// TIA Portal V20 export
// export: Created 2025-12-01T14:57:42.0271805Z, ExportSetting None, DisplayName Totally Integrated Automation Portal, DisplayVersion V20 Update 3, DisplayName TIA Portal Openness, DisplayVersion V20 Update 3, DisplayName TIA Portal Version Control Interface, DisplayVersion V20 Update 3, DisplayName STEP 7 Professional, DisplayVersion V20 Update 3, DisplayName STEP 7 Safety, DisplayVersion V20 Update 2, DisplayName WinCC Basic/Comfort/Advanced, DisplayVersion V20 Update 3, DisplayName WinCC Professional, DisplayVersion V20 Update 3, DisplayName WinCC Unified, DisplayVersion V20 Update 3
FUNCTION_BLOCK "FB382_HorquillaLenze_Paletizador_NDD_E3S3"   // FB382, LAD
{ S7_Optimized_Access := 'FALSE' }
// stored: AutoNumber false, SetENOAutomatically false
   VAR_INPUT
      Mesa : UInt;   // Mesa de la FB
      NDB_ConfigNDD : UInt;   // DB de Configuracion General del NDD
      NDB_DatosNDD : UInt;   // DB de Configuracion Particular del NDD
      OffsetDatosHorquilla : UInt;   // Offset de los datos particulares de la Horquilla
      DesHabilitar_Horq : Bool;   // DesHabilitar la Horquilla
      Mantenimiento : Bool;   // En Mantenimiento la Horquilla
      Error_Tx : Bool;   // Error de la Zona
      EnTension : Bool;   // Existe Tension en la Mesa
      TermicoFreno_Horq : Bool;   // Termico del Freno de la Horquilla
      Horq_PresCarga : Bool;   // Presencia de Carga en la Horquilla
      Horq_Protusion : Bool;
      Horq_SeguridadUp_Libre : Bool;
      Horq_SeguridadUp_Ocupada : Bool;
      Horq_SeguridadDown : Bool;
      BarreraNivelDown : Bool;
      EM_Horq_Out : Bool;   // Emergencia al Recoger la Horquilla
      Horq_Out : Bool;   // Horquilla Recogida
      Horq_In : Bool;   // Horquilla Fuera (En el Elevador)
      EM_Horq_In : Bool;   // Emergencia al Extender la Horquilla
      Manual_HorqIn : Bool;   // Extender la Horquilla en Manual
      Manual_HorqOut : Bool;   // Recoger la Horquilla en Manual
      Homming_Horq : Bool;   // Realizar el Homing del Variador de la Horquilla (RefCero >> Out)
      pHsRef_Horq : Bool;
      F_EnvMens_PMx : Bool;
      V_TOut_Horquilla : Time := T#5s;   // Valor de Time Out del Movimiento de la Horquilla
      V_TOut_Protusion : Time := T#500ms;
   END_VAR
   VAR_OUTPUT
      P_EnvMens_PMx : Bool;
   END_VAR
   VAR_IN_OUT
      Interlock_Horquilla : "NDD_Interlock_Horquilla";
   END_VAR
   VAR
      TOut_Horquilla { S7_SetPoint := 'True'} : TON_TIME;   // Time Out del Moviento de la Hoquilla
      TOut_Protusion { S7_SetPoint := 'True'} : TON_TIME;
      TEstableMovHorq { S7_SetPoint := 'True'} : TON_TIME;
      TEsperaMoverHorq { S7_SetPoint := 'True'} : TON_TIME;
      MemoPosicionActual_Horq : Int;
      PosicionActual_Horq : Int;   // Posicion Actual de la Horquilla (Variador)
      PosicionOut_Horq : Int;   // Posicion Out de la Horquilla (DB del NDD)
      PosicionIn_Horq { ExternalVisible := 'False'} : Int;   // Posicion In de la Horquilla (DB del NDD)
      PosicionMover_Horq : Int;
      ConsignaFR_Horq : Int;
      SubjectArea_Horq : Word;
      IDArea_Horq : Word;
      NodoNoPres_VarHorq : Bool;   // Nodo del Variador de la Horquilla - No presente
      MoverHorq : Bool;
      FinMoverHorq : Bool;
      MemoFinMorverHorq : Bool;
      PosHorqOut_OK : Bool;   // La Hoquilla esta en Reposo, esta en OUT
      PosHorqIn_OK : Bool;
      MA_Horquilla_IN : Bool;
      MA_Horquilla_OUT : Bool;
      HORQ_ET00 : Bool;   // Etapas de la Horquilla
      HORQ_ET01 : Bool;   // Etapas de la Horquilla
      HORQ_RST01 : Bool;   // Etapas de la Horquilla
      HORQ_RST02 : Bool;   // Etapas de la Horquilla
      HORQ_CAR01 : Bool;   // Etapas de la Horquilla
      HORQ_CAR02 : Bool;   // Etapas de la Horquilla
      HORQ_CAR03 : Bool;   // Etapas de la Horquilla
      HORQ_CAR04 : Bool;
      HORQ_ET02 : Bool;   // Etapas de la Horquilla
      HORQ_DCAR01 : Bool;   // Etapas de la Horquilla
      HORQ_DCAR02 : Bool;   // Etapas de la Horquilla
      HORQ_DCAR03 : Bool;   // Etapas de la Horquilla
      HORQ_DCAR04 : Bool;
      STAT_P_EnvMens_PMx : Bool;
      ErrorVar_Horquilla : Bool;
      ReferenciaOK_Horq : Bool;
      MemoReferenciaOK_Horq : Bool;
      MemoHoming_Horq : Bool;
   END_VAR
   VAR_TEMP
      EstadoZona : "EstadoZona";
      EstadoVI : "EstadosMesa_HorquillaLenze_Paletizador_NDD";
      NodoVar_Horq : "Status_NodosProfinet";
      Guardar_AR1 : DWord;
      Guardar_AR2 : DWord;
      P_DatosHorquilla : DWord;   // Puntero a los datos de la Horquilla (Configuracionn del Paletizador)
      P_NodoVar_Horq : DWord;
      DB_ConfigNDD : Word;   // DB de Configuracion General de los NDD
      DB_DatosNDD : Word;   // DB del NDD (Configuracion del Paletizador)
      NumDB_DiagProfinet : Word;
      NumNodo_VarHorq : Int;
      ByteInicial_VarHorq : Int;
      VeloManual_Horq : Int;   // Velocidad Manual
      VeloRapidaOut_Horq : Int;   // Velocidad Rapida para ir a Posicion Out
      VeloLentaOut_Horq : Int;   // Velocidad Lenta para ir a Posicion Out
      PosLentaOut_Horq : Int;   // Diferencia para pasar Lenta para ir a Posicion Out
      VeloRapidaIn_Horq : Int;   // Velocidad Rapida para ir a Posicion In
      VeloLentaIn_Horq : Int;   // Velocidad Lenta para ir a Posicion In
      PosLentaIn_Horq : Int;   // Diferencia para pasar Lenta para ir a Posicion In
      AuxMargen : Int;
      AuxPosMax : Int;
      AuxPosMin : Int;
      TempInt : Int;
      AuxEstados : Bool;
      DestinoHorq_OUT : Bool;
      DestinoHorq_IN : Bool;
      MoverHorq_LentaOUT : Bool;
      MoverHorq_LentaIN : Bool;
   END_VAR
   VAR_TEMP   // added for the SCL form of the ladder/FBD networks
      _w1 : Bool;
      _w2 : Bool;
      _w3 : Bool;
   END_VAR
BEGIN

REGION Network 1: INICIALIZACIONES
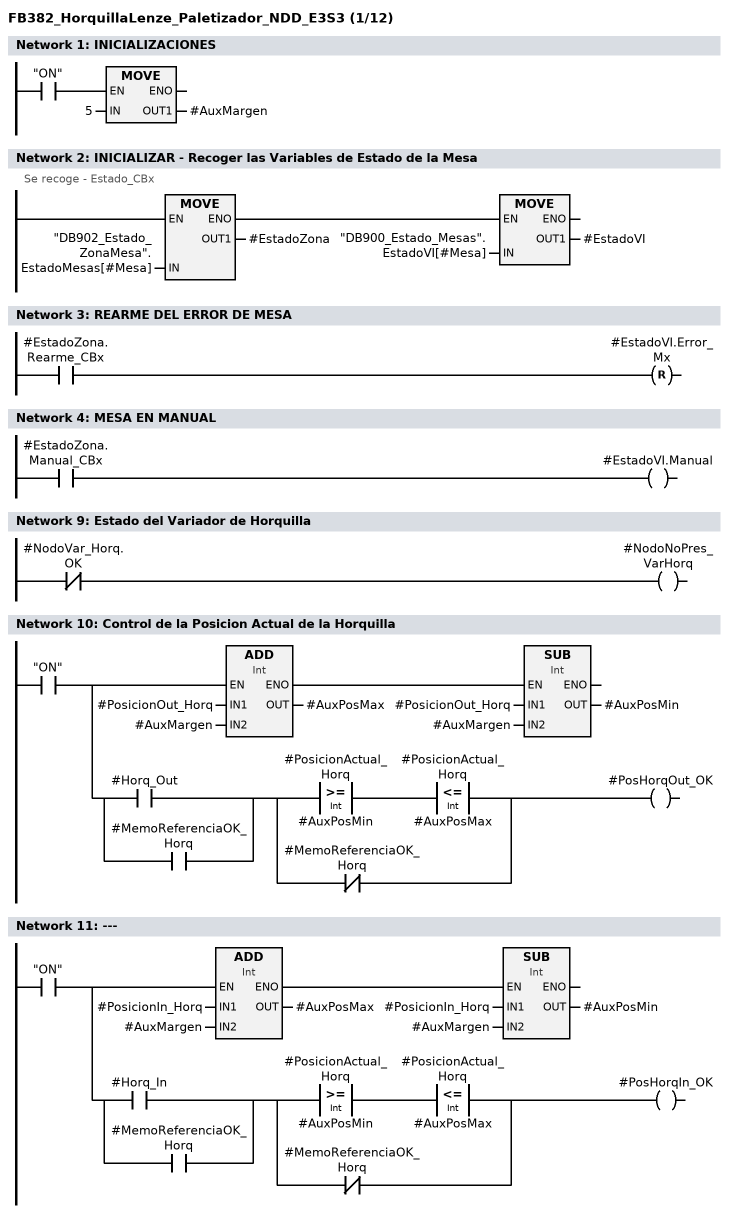
   RUNG wire#powerrail
      Contact( "ON" )
      { S7_GenerateENO := "TRUE" } Move(in := 5, out1 => #AuxMargen)
   END_RUNG
   // the same network as SCL:
   IF "ON" THEN #AuxMargen := 5; END_IF;
END_REGION

REGION Network 2: INICIALIZAR - Recoger las Variables de Estado de la Mesa
   // Se recoge - Estado_CBx
   RUNG wire#powerrail
      Move(in := "DB902_Estado_ZonaMesa".EstadoMesas[#Mesa], out1 => #EstadoZona)
      Move(in := "DB900_Estado_Mesas".EstadoVI[#Mesa], out1 => #EstadoVI)
   END_RUNG
   // the same network as SCL:
   #EstadoZona := "DB902_Estado_ZonaMesa".EstadoMesas[#Mesa];
   #EstadoVI := "DB900_Estado_Mesas".EstadoVI[#Mesa];
END_REGION

REGION Network 3: REARME DEL ERROR DE MESA
   RUNG wire#powerrail
      Contact( #EstadoZona.Rearme_CBx )
      R_Coil( #EstadoVI.Error_Mx )
   END_RUNG
   // the same network as SCL:
   IF #EstadoZona.Rearme_CBx THEN #EstadoVI.Error_Mx := FALSE; END_IF;
END_REGION

REGION Network 4: MESA EN MANUAL
   RUNG wire#powerrail
      Contact( #EstadoZona.Manual_CBx )
      Coil( #EstadoVI.Manual )
   END_RUNG
   // the same network as SCL:
   #EstadoVI.Manual := #EstadoZona.Manual_CBx;
END_REGION

NETWORK
TITLE = Datos Internos de la Horquilla
// ------------------------------------------------------------------------------------
// ------------------------------------------------------------------------------------
// --- Previas

      TAR1  #Guardar_AR1;  // Guardar AR1 y AR2


// ------------------------------------------------------------------------------------
// ------------------------------------------------------------------------------------
// --- Datos iniciales

      L     #NDB_DatosNDD;  // - DB del Paletizador NDD
      T     #DB_DatosNDD;

      L     #NDB_ConfigNDD;  // - DB del Config de los Paletizadores MDD
      T     #DB_ConfigNDD;  //

      L     #OffsetDatosHorquilla;  // Puntero a los Datos de Horquilla
      SLD   3;
      T     #P_DatosHorquilla;


/////////////////////////////////////////////////////////////////////////////
/////////////////////////////////////////////////////////////////////////////
// --- Sistema de Profinet

      LAR1  P#0.0;  // - Leer Datos de los Variadores
      OPN   DB [#DB_DatosNDD];  //   del NDD

      L     DBW [AR1, P#0.0];  // - Num DB de Profinet
      T     #NumDB_DiagProfinet;
      L     DBW [AR1, P#6.0];  // - Nodos de los Variadores
      T     #NumNodo_VarHorq;
      L     DBW [AR1, P#12.0];  // - Direcciones de los Variadores
      T     #ByteInicial_VarHorq;

      L     P##NodoVar_Horq;  // Puntero del Estado del Nodo del Variador de Horquilla (TEMPORAL)
      T     #P_NodoVar_Horq;



NETWORK
TITLE = ---
// ------------------------------------------------------------------------------------
// ------------------------------------------------------------------------------------
// --- Datos Generales de Configuracion de los NDD

      LAR1  P#0.0;  // - Leer Datos de Velocidad de la Horquilla
      OPN   DB [#DB_ConfigNDD];

      L     DBW [AR1, P#16.0];  // - Velocidad en Manual
      T     #VeloManual_Horq;

      L     DBW [AR1, P#18.0];  // - Velocidad del Mov. hacia In
      T     #VeloRapidaIn_Horq;
      L     DBW [AR1, P#20.0];
      T     #VeloLentaIn_Horq;

      L     DBW [AR1, P#22.0];  // - Velocidad del Mov. hacia Out
      T     #VeloRapidaOut_Horq;
      L     DBW [AR1, P#24.0];
      T     #VeloLentaOut_Horq;

      L     DBW [AR1, P#26.0];  // - Posiciones de Cambio de Velocidad
      T     #PosLentaIn_Horq;
      L     DBW [AR1, P#28.0];
      T     #PosLentaOut_Horq;



NETWORK
TITLE = ----
// ------------------------------------------------------------------------------------
// ------------------------------------------------------------------------------------
// --- Datos Particulares de la Horquilla del NDD

      LAR1  #P_DatosHorquilla;  // - Leer Datos de la Horquilla
      OPN   DB [#DB_DatosNDD];
      L     DBW [AR1, P#0.0];
      T     #PosicionIn_Horq;
      L     DBW [AR1, P#2.0];
      T     #PosicionOut_Horq;


// ------------------------------------------------------------------------------------
// ------------------------------------------------------------------------------------
// --- Estado del Nodo de PROFINET del Variador de la Horquilla (LENZE)

      L     #NumNodo_VarHorq;  // Nodo de Profinet
      L     1;
      -I;
      L     2;  // Longitud registro datos
      *I;
      SLD   3;
      LAR1;

      OPN   DB [#NumDB_DiagProfinet];  // Leer estado del Nodo de PROFINET
      L     DBW [AR1, P#0.0];
      T     LW [#P_NodoVar_Horq];




NETWORK
TITLE = ---
// ------------------------------------------------------------------------------------
// ------------------------------------------------------------------------------------
// --- Final de Datos Inicialies

      LAR1  #Guardar_AR1;  // Recuperar AR1 y AR2



REGION Network 9: Estado del Variador de Horquilla
   RUNG wire#powerrail
      I_Contact( #NodoVar_Horq.OK )
      Coil( #NodoNoPres_VarHorq )
   END_RUNG
   // the same network as SCL:
   #NodoNoPres_VarHorq := NOT #NodoVar_Horq.OK;
END_REGION

REGION Network 10: Control de la Posicion Actual de la Horquilla
   RUNG wire#powerrail
      Contact( "ON" )
      wire#w1
      { S7_Templates := "SrcType := Int"; S7_GenerateENO := "TRUE" } Add(in1 := #PosicionOut_Horq, in2 := #AuxMargen, out => #AuxPosMax)
      { S7_Templates := "SrcType := Int"; S7_GenerateENO := "TRUE" } Sub(in1 := #PosicionOut_Horq, in2 := #AuxMargen, out => #AuxPosMin)
   END_RUNG
   RUNG wire#w1
      Contact( #Horq_Out )
      wire#w2
      { S7_Templates := "SrcType := Int" } GE_Contact(in1 := #PosicionActual_Horq, in2 := #AuxPosMin)
      { S7_Templates := "SrcType := Int" } LE_Contact(in1 := #PosicionActual_Horq, in2 := #AuxPosMax)
      wire#w3
      Coil( #PosHorqOut_OK )
   END_RUNG
   RUNG wire#w1
      Contact( #MemoReferenciaOK_Horq )
   END_RUNG wire#w2
   RUNG wire#w2
      I_Contact( #MemoReferenciaOK_Horq )
   END_RUNG wire#w3
   // the same network as SCL:
   // ENO of a box is taken as its EN; it also drops when the box reports an error
   IF "ON" THEN
       #AuxPosMax := #PosicionOut_Horq + #AuxMargen;
       #AuxPosMin := #PosicionOut_Horq - #AuxMargen;
   END_IF;
   #PosHorqOut_OK := "ON" AND (#Horq_Out OR #MemoReferenciaOK_Horq) AND (((#PosicionActual_Horq >= #AuxPosMin) AND (#PosicionActual_Horq <= #AuxPosMax)) OR NOT #MemoReferenciaOK_Horq);
END_REGION

REGION Network 11: ---
   RUNG wire#powerrail
      Contact( "ON" )
      wire#w1
      { S7_Templates := "SrcType := Int"; S7_GenerateENO := "TRUE" } Add(in1 := #PosicionIn_Horq, in2 := #AuxMargen, out => #AuxPosMax)
      { S7_Templates := "SrcType := Int"; S7_GenerateENO := "TRUE" } Sub(in1 := #PosicionIn_Horq, in2 := #AuxMargen, out => #AuxPosMin)
   END_RUNG
   RUNG wire#w1
      Contact( #Horq_In )
      wire#w2
      { S7_Templates := "SrcType := Int" } GE_Contact(in1 := #PosicionActual_Horq, in2 := #AuxPosMin)
      { S7_Templates := "SrcType := Int" } LE_Contact(in1 := #PosicionActual_Horq, in2 := #AuxPosMax)
      wire#w3
      Coil( #PosHorqIn_OK )
   END_RUNG
   RUNG wire#w1
      Contact( #MemoReferenciaOK_Horq )
   END_RUNG wire#w2
   RUNG wire#w2
      I_Contact( #MemoReferenciaOK_Horq )
   END_RUNG wire#w3
   // the same network as SCL:
   // ENO of a box is taken as its EN; it also drops when the box reports an error
   IF "ON" THEN
       #AuxPosMax := #PosicionIn_Horq + #AuxMargen;
       #AuxPosMin := #PosicionIn_Horq - #AuxMargen;
   END_IF;
   #PosHorqIn_OK := "ON" AND (#Horq_In OR #MemoReferenciaOK_Horq) AND (((#PosicionActual_Horq >= #AuxPosMin) AND (#PosicionActual_Horq <= #AuxPosMax)) OR NOT #MemoReferenciaOK_Horq);
END_REGION

REGION Network 12: ---
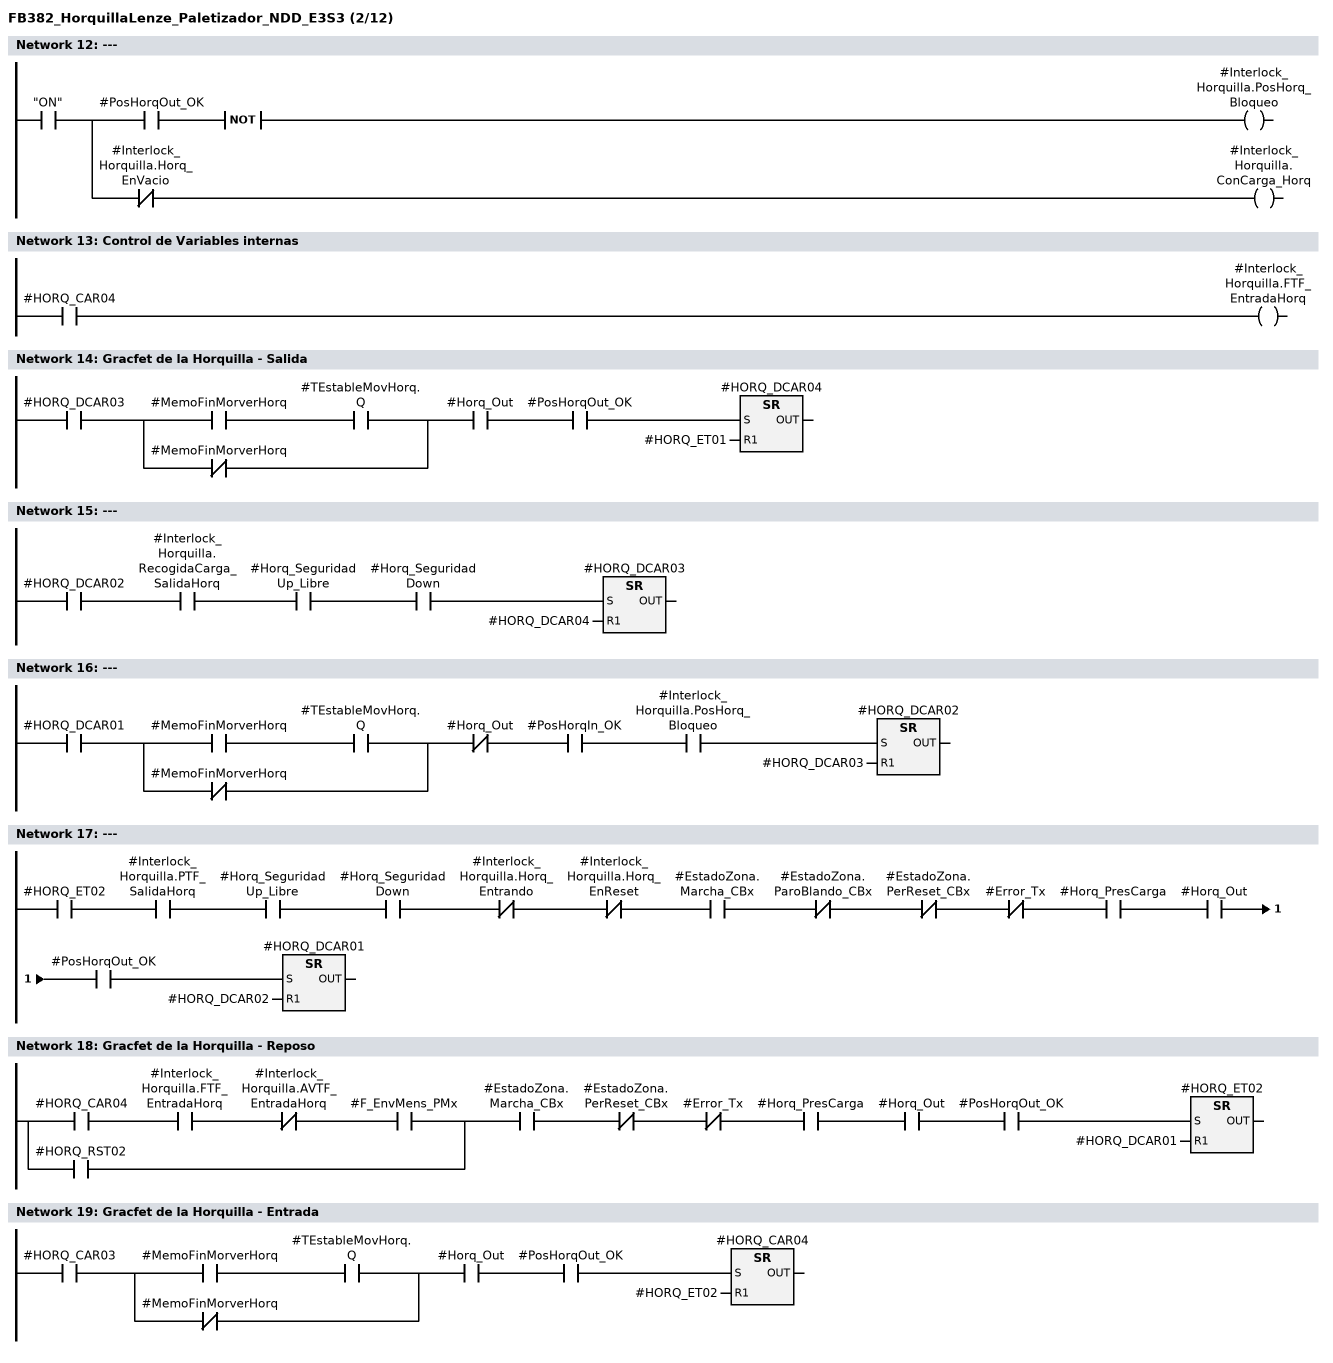
   RUNG wire#powerrail
      Contact( "ON" )
      wire#w1
      Contact( #PosHorqOut_OK )
      Not()
      Coil( #Interlock_Horquilla.PosHorq_Bloqueo )
   END_RUNG
   RUNG wire#w1
      I_Contact( #Interlock_Horquilla.Horq_EnVacio )
      Coil( #Interlock_Horquilla.ConCarga_Horq )
   END_RUNG
   // the same network as SCL:
   #Interlock_Horquilla.PosHorq_Bloqueo := NOT ("ON" AND #PosHorqOut_OK);
   #Interlock_Horquilla.ConCarga_Horq := "ON" AND NOT #Interlock_Horquilla.Horq_EnVacio;
END_REGION

REGION Network 13: Control de Variables internas
   RUNG wire#powerrail
      Contact( #HORQ_CAR04 )
      Coil( #Interlock_Horquilla.FTF_EntradaHorq )
   END_RUNG
   // the same network as SCL:
   #Interlock_Horquilla.FTF_EntradaHorq := #HORQ_CAR04;
END_REGION

REGION Network 14: Gracfet de la Horquilla - Salida
   RUNG wire#powerrail
      Contact( #HORQ_DCAR03 )
      wire#w1
      Contact( #MemoFinMorverHorq )
      Contact( #TEstableMovHorq.Q )
      wire#w2
      Contact( #Horq_Out )
      Contact( #PosHorqOut_OK )
      S_SR(operand := #HORQ_DCAR04, r1 := #HORQ_ET01)
   END_RUNG
   RUNG wire#w1
      I_Contact( #MemoFinMorverHorq )
   END_RUNG wire#w2
   // the same network as SCL:
   IF #HORQ_DCAR03 AND ((#MemoFinMorverHorq AND #TEstableMovHorq.Q) OR NOT #MemoFinMorverHorq) AND #Horq_Out AND #PosHorqOut_OK THEN
       #HORQ_DCAR04 := TRUE;   // SR flip-flop
   END_IF;
   IF #HORQ_ET01 THEN #HORQ_DCAR04 := FALSE; END_IF;
END_REGION

REGION Network 15: ---
   RUNG wire#powerrail
      Contact( #HORQ_DCAR02 )
      Contact( #Interlock_Horquilla.RecogidaCarga_SalidaHorq )
      Contact( #Horq_SeguridadUp_Libre )
      Contact( #Horq_SeguridadDown )
      S_SR(operand := #HORQ_DCAR03, r1 := #HORQ_DCAR04)
   END_RUNG
   // the same network as SCL:
   IF #HORQ_DCAR02 AND #Interlock_Horquilla.RecogidaCarga_SalidaHorq AND #Horq_SeguridadUp_Libre AND #Horq_SeguridadDown THEN
       #HORQ_DCAR03 := TRUE;   // SR flip-flop
   END_IF;
   IF #HORQ_DCAR04 THEN #HORQ_DCAR03 := FALSE; END_IF;
END_REGION

REGION Network 16: ---
   RUNG wire#powerrail
      Contact( #HORQ_DCAR01 )
      wire#w1
      Contact( #MemoFinMorverHorq )
      Contact( #TEstableMovHorq.Q )
      wire#w2
      I_Contact( #Horq_Out )
      Contact( #PosHorqIn_OK )
      Contact( #Interlock_Horquilla.PosHorq_Bloqueo )
      S_SR(operand := #HORQ_DCAR02, r1 := #HORQ_DCAR03)
   END_RUNG
   RUNG wire#w1
      I_Contact( #MemoFinMorverHorq )
   END_RUNG wire#w2
   // the same network as SCL:
   IF #HORQ_DCAR01 AND ((#MemoFinMorverHorq AND #TEstableMovHorq.Q) OR NOT #MemoFinMorverHorq) AND NOT #Horq_Out AND #PosHorqIn_OK AND #Interlock_Horquilla.PosHorq_Bloqueo THEN
       #HORQ_DCAR02 := TRUE;   // SR flip-flop
   END_IF;
   IF #HORQ_DCAR03 THEN #HORQ_DCAR02 := FALSE; END_IF;
END_REGION

REGION Network 17: ---
   RUNG wire#powerrail
      Contact( #HORQ_ET02 )
      Contact( #Interlock_Horquilla.PTF_SalidaHorq )
      Contact( #Horq_SeguridadUp_Libre )
      Contact( #Horq_SeguridadDown )
      I_Contact( #Interlock_Horquilla.Horq_Entrando )
      I_Contact( #Interlock_Horquilla.Horq_EnReset )
      Contact( #EstadoZona.Marcha_CBx )
      I_Contact( #EstadoZona.ParoBlando_CBx )
      I_Contact( #EstadoZona.PerReset_CBx )
      I_Contact( #Error_Tx )
      Contact( #Horq_PresCarga )
      Contact( #Horq_Out )
      Contact( #PosHorqOut_OK )
      S_SR(operand := #HORQ_DCAR01, r1 := #HORQ_DCAR02)
   END_RUNG
   // the same network as SCL:
   IF #HORQ_ET02 AND #Interlock_Horquilla.PTF_SalidaHorq AND #Horq_SeguridadUp_Libre AND #Horq_SeguridadDown AND NOT #Interlock_Horquilla.Horq_Entrando AND NOT #Interlock_Horquilla.Horq_EnReset AND #EstadoZona.Marcha_CBx AND NOT #EstadoZona.ParoBlando_CBx AND NOT #EstadoZona.PerReset_CBx AND NOT #Error_Tx AND #Horq_PresCarga AND #Horq_Out AND #PosHorqOut_OK THEN
       #HORQ_DCAR01 := TRUE;   // SR flip-flop
   END_IF;
   IF #HORQ_DCAR02 THEN #HORQ_DCAR01 := FALSE; END_IF;
END_REGION

REGION Network 18: Gracfet de la Horquilla - Reposo
   RUNG wire#powerrail
      Contact( #HORQ_CAR04 )
      Contact( #Interlock_Horquilla.FTF_EntradaHorq )
      I_Contact( #Interlock_Horquilla.AVTF_EntradaHorq )
      Contact( #F_EnvMens_PMx )
      wire#w1
      Contact( #EstadoZona.Marcha_CBx )
      I_Contact( #EstadoZona.PerReset_CBx )
      I_Contact( #Error_Tx )
      Contact( #Horq_PresCarga )
      Contact( #Horq_Out )
      Contact( #PosHorqOut_OK )
      S_SR(operand := #HORQ_ET02, r1 := #HORQ_DCAR01)
   END_RUNG
   RUNG wire#powerrail
      Contact( #HORQ_RST02 )
   END_RUNG wire#w1
   // the same network as SCL:
   IF ((#HORQ_CAR04 AND #Interlock_Horquilla.FTF_EntradaHorq AND NOT #Interlock_Horquilla.AVTF_EntradaHorq AND #F_EnvMens_PMx) OR #HORQ_RST02) AND #EstadoZona.Marcha_CBx AND NOT #EstadoZona.PerReset_CBx AND NOT #Error_Tx AND #Horq_PresCarga AND #Horq_Out AND #PosHorqOut_OK THEN
       #HORQ_ET02 := TRUE;   // SR flip-flop
   END_IF;
   IF #HORQ_DCAR01 THEN #HORQ_ET02 := FALSE; END_IF;
END_REGION

REGION Network 19: Gracfet de la Horquilla - Entrada
   RUNG wire#powerrail
      Contact( #HORQ_CAR03 )
      wire#w1
      Contact( #MemoFinMorverHorq )
      Contact( #TEstableMovHorq.Q )
      wire#w2
      Contact( #Horq_Out )
      Contact( #PosHorqOut_OK )
      S_SR(operand := #HORQ_CAR04, r1 := #HORQ_ET02)
   END_RUNG
   RUNG wire#w1
      I_Contact( #MemoFinMorverHorq )
   END_RUNG wire#w2
   // the same network as SCL:
   IF #HORQ_CAR03 AND ((#MemoFinMorverHorq AND #TEstableMovHorq.Q) OR NOT #MemoFinMorverHorq) AND #Horq_Out AND #PosHorqOut_OK THEN
       #HORQ_CAR04 := TRUE;   // SR flip-flop
   END_IF;
   IF #HORQ_ET02 THEN #HORQ_CAR04 := FALSE; END_IF;
END_REGION

REGION Network 20: ---
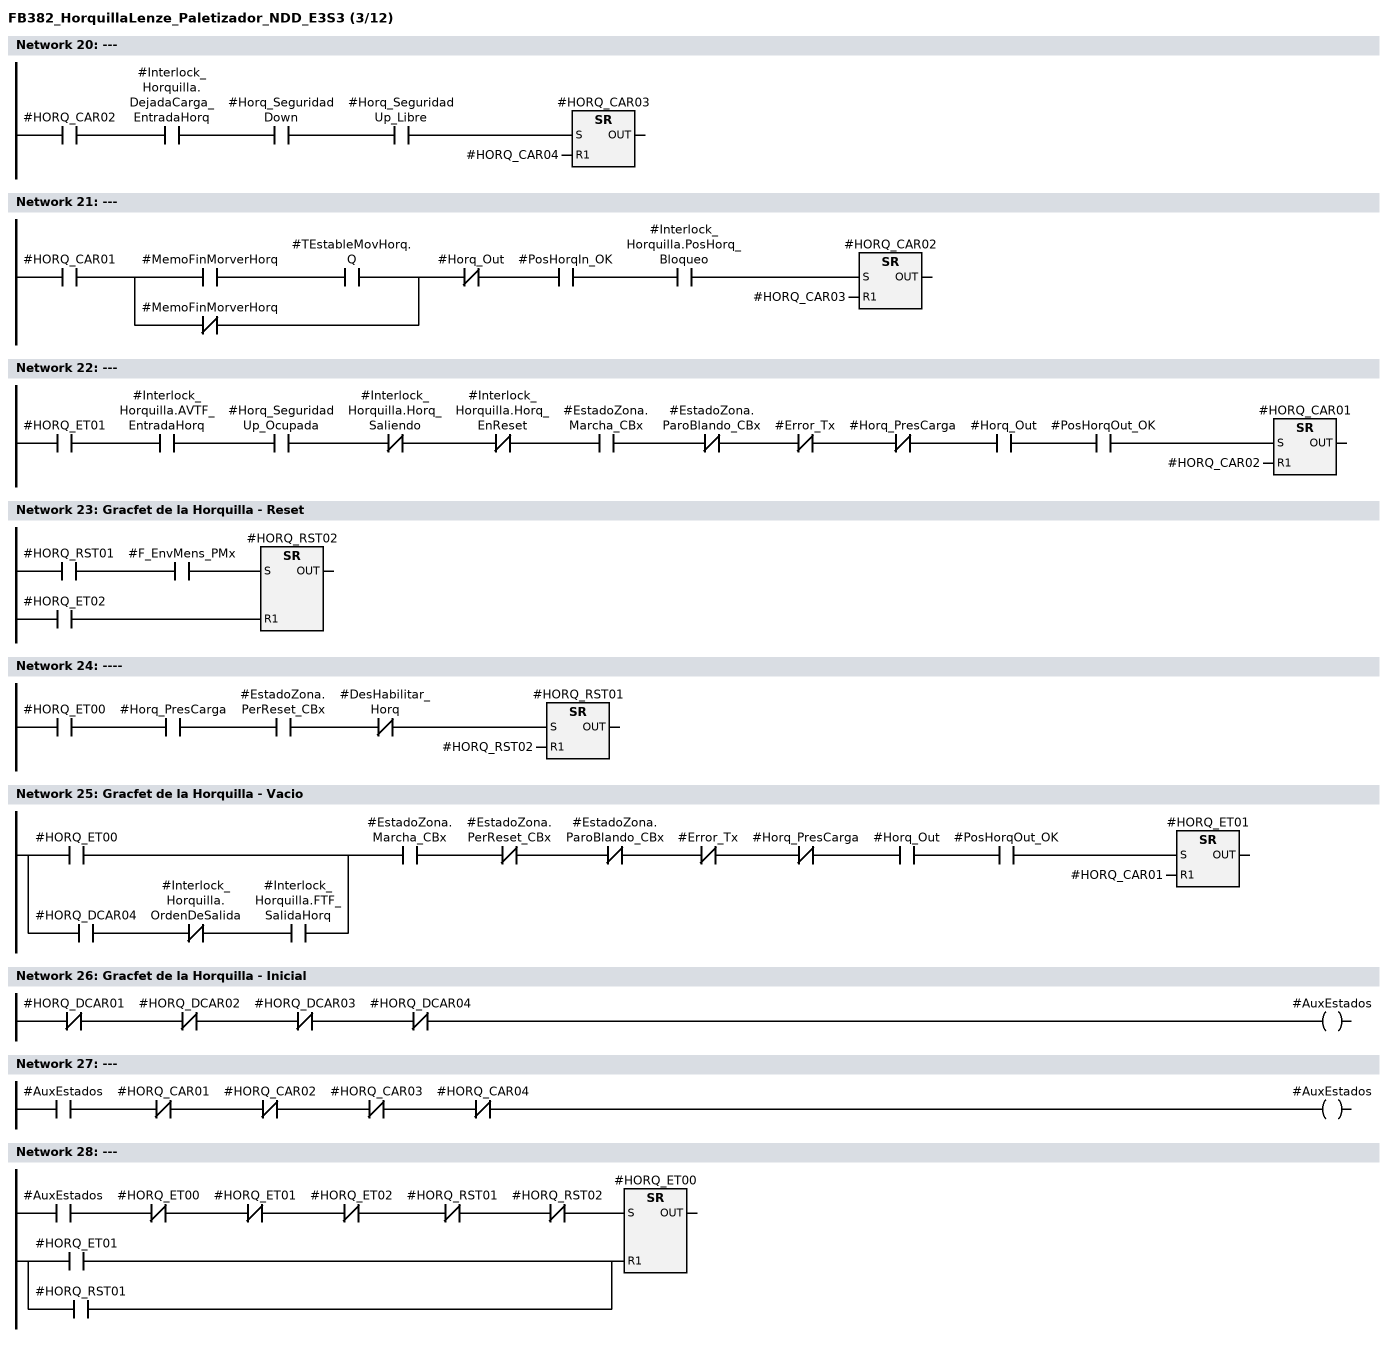
   RUNG wire#powerrail
      Contact( #HORQ_CAR02 )
      Contact( #Interlock_Horquilla.DejadaCarga_EntradaHorq )
      Contact( #Horq_SeguridadDown )
      Contact( #Horq_SeguridadUp_Libre )
      S_SR(operand := #HORQ_CAR03, r1 := #HORQ_CAR04)
   END_RUNG
   // the same network as SCL:
   IF #HORQ_CAR02 AND #Interlock_Horquilla.DejadaCarga_EntradaHorq AND #Horq_SeguridadDown AND #Horq_SeguridadUp_Libre THEN
       #HORQ_CAR03 := TRUE;   // SR flip-flop
   END_IF;
   IF #HORQ_CAR04 THEN #HORQ_CAR03 := FALSE; END_IF;
END_REGION

REGION Network 21: ---
   RUNG wire#powerrail
      Contact( #HORQ_CAR01 )
      wire#w1
      Contact( #MemoFinMorverHorq )
      Contact( #TEstableMovHorq.Q )
      wire#w2
      I_Contact( #Horq_Out )
      Contact( #PosHorqIn_OK )
      Contact( #Interlock_Horquilla.PosHorq_Bloqueo )
      S_SR(operand := #HORQ_CAR02, r1 := #HORQ_CAR03)
   END_RUNG
   RUNG wire#w1
      I_Contact( #MemoFinMorverHorq )
   END_RUNG wire#w2
   // the same network as SCL:
   IF #HORQ_CAR01 AND ((#MemoFinMorverHorq AND #TEstableMovHorq.Q) OR NOT #MemoFinMorverHorq) AND NOT #Horq_Out AND #PosHorqIn_OK AND #Interlock_Horquilla.PosHorq_Bloqueo THEN
       #HORQ_CAR02 := TRUE;   // SR flip-flop
   END_IF;
   IF #HORQ_CAR03 THEN #HORQ_CAR02 := FALSE; END_IF;
END_REGION

REGION Network 22: ---
   RUNG wire#powerrail
      Contact( #HORQ_ET01 )
      Contact( #Interlock_Horquilla.AVTF_EntradaHorq )
      Contact( #Horq_SeguridadUp_Ocupada )
      I_Contact( #Interlock_Horquilla.Horq_Saliendo )
      I_Contact( #Interlock_Horquilla.Horq_EnReset )
      Contact( #EstadoZona.Marcha_CBx )
      I_Contact( #EstadoZona.ParoBlando_CBx )
      I_Contact( #Error_Tx )
      I_Contact( #Horq_PresCarga )
      Contact( #Horq_Out )
      Contact( #PosHorqOut_OK )
      S_SR(operand := #HORQ_CAR01, r1 := #HORQ_CAR02)
   END_RUNG
   // the same network as SCL:
   IF #HORQ_ET01 AND #Interlock_Horquilla.AVTF_EntradaHorq AND #Horq_SeguridadUp_Ocupada AND NOT #Interlock_Horquilla.Horq_Saliendo AND NOT #Interlock_Horquilla.Horq_EnReset AND #EstadoZona.Marcha_CBx AND NOT #EstadoZona.ParoBlando_CBx AND NOT #Error_Tx AND NOT #Horq_PresCarga AND #Horq_Out AND #PosHorqOut_OK THEN
       #HORQ_CAR01 := TRUE;   // SR flip-flop
   END_IF;
   IF #HORQ_CAR02 THEN #HORQ_CAR01 := FALSE; END_IF;
END_REGION

REGION Network 23: Gracfet de la Horquilla - Reset
   RUNG wire#powerrail
      Contact( #HORQ_RST01 )
      Contact( #F_EnvMens_PMx )
      S_SR(operand := #HORQ_RST02, r1 := wire#w1)
   END_RUNG
   RUNG wire#powerrail
      Contact( #HORQ_ET02 )
   END_RUNG wire#w1
   // the same network as SCL:
   IF #HORQ_RST01 AND #F_EnvMens_PMx THEN
       #HORQ_RST02 := TRUE;   // SR flip-flop
   END_IF;
   IF #HORQ_ET02 THEN #HORQ_RST02 := FALSE; END_IF;
END_REGION

REGION Network 24: ----
   RUNG wire#powerrail
      Contact( #HORQ_ET00 )
      Contact( #Horq_PresCarga )
      Contact( #EstadoZona.PerReset_CBx )
      I_Contact( #DesHabilitar_Horq )
      S_SR(operand := #HORQ_RST01, r1 := #HORQ_RST02)
   END_RUNG
   // the same network as SCL:
   IF #HORQ_ET00 AND #Horq_PresCarga AND #EstadoZona.PerReset_CBx AND NOT #DesHabilitar_Horq THEN
       #HORQ_RST01 := TRUE;   // SR flip-flop
   END_IF;
   IF #HORQ_RST02 THEN #HORQ_RST01 := FALSE; END_IF;
END_REGION

REGION Network 25: Gracfet de la Horquilla - Vacio
   RUNG wire#powerrail
      Contact( #HORQ_ET00 )
      wire#w1
      Contact( #EstadoZona.Marcha_CBx )
      I_Contact( #EstadoZona.PerReset_CBx )
      I_Contact( #EstadoZona.ParoBlando_CBx )
      I_Contact( #Error_Tx )
      I_Contact( #Horq_PresCarga )
      Contact( #Horq_Out )
      Contact( #PosHorqOut_OK )
      S_SR(operand := #HORQ_ET01, r1 := #HORQ_CAR01)
   END_RUNG
   RUNG wire#powerrail
      Contact( #HORQ_DCAR04 )
      I_Contact( #Interlock_Horquilla.OrdenDeSalida )
      Contact( #Interlock_Horquilla.FTF_SalidaHorq )
   END_RUNG wire#w1
   // the same network as SCL:
   IF (#HORQ_ET00 OR (#HORQ_DCAR04 AND NOT #Interlock_Horquilla.OrdenDeSalida AND #Interlock_Horquilla.FTF_SalidaHorq)) AND #EstadoZona.Marcha_CBx AND NOT #EstadoZona.PerReset_CBx AND NOT #EstadoZona.ParoBlando_CBx AND NOT #Error_Tx AND NOT #Horq_PresCarga AND #Horq_Out AND #PosHorqOut_OK THEN
       #HORQ_ET01 := TRUE;   // SR flip-flop
   END_IF;
   IF #HORQ_CAR01 THEN #HORQ_ET01 := FALSE; END_IF;
END_REGION

REGION Network 26: Gracfet de la Horquilla - Inicial
   RUNG wire#powerrail
      I_Contact( #HORQ_DCAR01 )
      I_Contact( #HORQ_DCAR02 )
      I_Contact( #HORQ_DCAR03 )
      I_Contact( #HORQ_DCAR04 )
      Coil( #AuxEstados )
   END_RUNG
   // the same network as SCL:
   #AuxEstados := NOT #HORQ_DCAR01 AND NOT #HORQ_DCAR02 AND NOT #HORQ_DCAR03 AND NOT #HORQ_DCAR04;
END_REGION

REGION Network 27: ---
   RUNG wire#powerrail
      Contact( #AuxEstados )
      I_Contact( #HORQ_CAR01 )
      I_Contact( #HORQ_CAR02 )
      I_Contact( #HORQ_CAR03 )
      I_Contact( #HORQ_CAR04 )
      Coil( #AuxEstados )
   END_RUNG
   // the same network as SCL:
   #AuxEstados := #AuxEstados AND NOT #HORQ_CAR01 AND NOT #HORQ_CAR02 AND NOT #HORQ_CAR03 AND NOT #HORQ_CAR04;
END_REGION

REGION Network 28: ---
   RUNG wire#powerrail
      Contact( #AuxEstados )
      I_Contact( #HORQ_ET00 )
      I_Contact( #HORQ_ET01 )
      I_Contact( #HORQ_ET02 )
      I_Contact( #HORQ_RST01 )
      I_Contact( #HORQ_RST02 )
      S_SR(operand := #HORQ_ET00, r1 := wire#w1)
   END_RUNG
   RUNG wire#powerrail
      Contact( #HORQ_ET01 )
   END_RUNG wire#w1
   RUNG wire#powerrail
      Contact( #HORQ_RST01 )
   END_RUNG wire#w1
   // the same network as SCL:
   IF #AuxEstados AND NOT #HORQ_ET00 AND NOT #HORQ_ET01 AND NOT #HORQ_ET02 AND NOT #HORQ_RST01 AND NOT #HORQ_RST02 THEN
       #HORQ_ET00 := TRUE;   // SR flip-flop
   END_IF;
   IF #HORQ_ET01 OR #HORQ_RST01 THEN #HORQ_ET00 := FALSE; END_IF;
END_REGION

REGION Network 29: Fin Reset y Fin Paro Blando
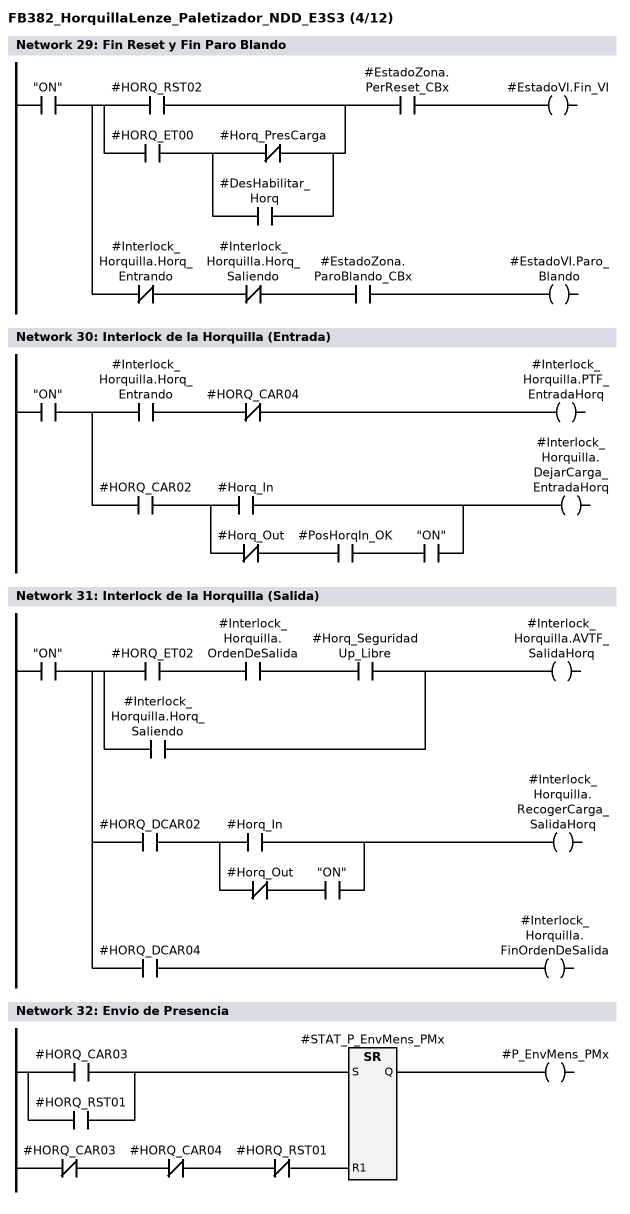
   RUNG wire#powerrail
      Contact( "ON" )
      wire#w1
      Contact( #HORQ_RST02 )
      wire#w2
      Contact( #EstadoZona.PerReset_CBx )
      Coil( #EstadoVI.Fin_VI )
   END_RUNG
   RUNG wire#w1
      Contact( #HORQ_ET00 )
      wire#w3
      I_Contact( #Horq_PresCarga )
   END_RUNG wire#w2
   RUNG wire#w3
      Contact( #DesHabilitar_Horq )
   END_RUNG wire#w2
   RUNG wire#w1
      I_Contact( #Interlock_Horquilla.Horq_Entrando )
      I_Contact( #Interlock_Horquilla.Horq_Saliendo )
      Contact( #EstadoZona.ParoBlando_CBx )
      Coil( #EstadoVI.Paro_Blando )
   END_RUNG
   // the same network as SCL:
   #EstadoVI.Fin_VI := "ON" AND (#HORQ_RST02 OR (#HORQ_ET00 AND (NOT #Horq_PresCarga OR #DesHabilitar_Horq))) AND #EstadoZona.PerReset_CBx;
   #EstadoVI.Paro_Blando := "ON" AND NOT #Interlock_Horquilla.Horq_Entrando AND NOT #Interlock_Horquilla.Horq_Saliendo AND #EstadoZona.ParoBlando_CBx;
END_REGION

REGION Network 30: Interlock de la Horquilla (Entrada)
   RUNG wire#powerrail
      Contact( "ON" )
      wire#w1
      Contact( #Interlock_Horquilla.Horq_Entrando )
      I_Contact( #HORQ_CAR04 )
      Coil( #Interlock_Horquilla.PTF_EntradaHorq )
   END_RUNG
   RUNG wire#w1
      Contact( #HORQ_CAR02 )
      wire#w2
      Contact( #Horq_In )
      wire#w3
      Coil( #Interlock_Horquilla.DejarCarga_EntradaHorq )
   END_RUNG
   RUNG wire#w2
      I_Contact( #Horq_Out )
      Contact( #PosHorqIn_OK )
      Contact( "ON" )
   END_RUNG wire#w3
   // the same network as SCL:
   #Interlock_Horquilla.PTF_EntradaHorq := "ON" AND #Interlock_Horquilla.Horq_Entrando AND NOT #HORQ_CAR04;
   #Interlock_Horquilla.DejarCarga_EntradaHorq := "ON" AND #HORQ_CAR02 AND (#Horq_In OR (NOT #Horq_Out AND #PosHorqIn_OK AND "ON"));
END_REGION

REGION Network 31: Interlock de la Horquilla (Salida)
   RUNG wire#powerrail
      Contact( "ON" )
      wire#w1
      Contact( #HORQ_ET02 )
      Contact( #Interlock_Horquilla.OrdenDeSalida )
      Contact( #Horq_SeguridadUp_Libre )
      wire#w2
      Coil( #Interlock_Horquilla.AVTF_SalidaHorq )
   END_RUNG
   RUNG wire#w1
      Contact( #Interlock_Horquilla.Horq_Saliendo )
   END_RUNG wire#w2
   RUNG wire#w1
      Contact( #HORQ_DCAR02 )
      wire#w3
      Contact( #Horq_In )
      wire#w4
      Coil( #Interlock_Horquilla.RecogerCarga_SalidaHorq )
   END_RUNG
   RUNG wire#w3
      I_Contact( #Horq_Out )
      Contact( "ON" )
   END_RUNG wire#w4
   RUNG wire#w1
      Contact( #HORQ_DCAR04 )
      Coil( #Interlock_Horquilla.FinOrdenDeSalida )
   END_RUNG
   // the same network as SCL:
   #Interlock_Horquilla.AVTF_SalidaHorq := "ON" AND ((#HORQ_ET02 AND #Interlock_Horquilla.OrdenDeSalida AND #Horq_SeguridadUp_Libre) OR #Interlock_Horquilla.Horq_Saliendo);
   #Interlock_Horquilla.RecogerCarga_SalidaHorq := "ON" AND #HORQ_DCAR02 AND (#Horq_In OR (NOT #Horq_Out AND "ON"));
   #Interlock_Horquilla.FinOrdenDeSalida := "ON" AND #HORQ_DCAR04;
END_REGION

REGION Network 32: Envio de Presencia
   RUNG wire#powerrail
      Contact( #HORQ_CAR03 )
      wire#w1
      S_SR(operand := #STAT_P_EnvMens_PMx, r1 := wire#w2)
      Coil( #P_EnvMens_PMx )
   END_RUNG
   RUNG wire#powerrail
      Contact( #HORQ_RST01 )
   END_RUNG wire#w1
   RUNG wire#powerrail
      I_Contact( #HORQ_CAR03 )
      I_Contact( #HORQ_CAR04 )
      I_Contact( #HORQ_RST01 )
   END_RUNG wire#w2
   // the same network as SCL:
   IF #HORQ_CAR03 OR #HORQ_RST01 THEN
       #STAT_P_EnvMens_PMx := TRUE;   // SR flip-flop
   END_IF;
   IF NOT #HORQ_CAR03 AND NOT #HORQ_CAR04 AND NOT #HORQ_RST01 THEN #STAT_P_EnvMens_PMx := FALSE; END_IF;
   #P_EnvMens_PMx := #STAT_P_EnvMens_PMx;
END_REGION

REGION Network 33: Control - Movimiento de la Horquilla En Semi-Automatico
   // Cuidado sino tiene Referencia tambien se mueve (En Lento)
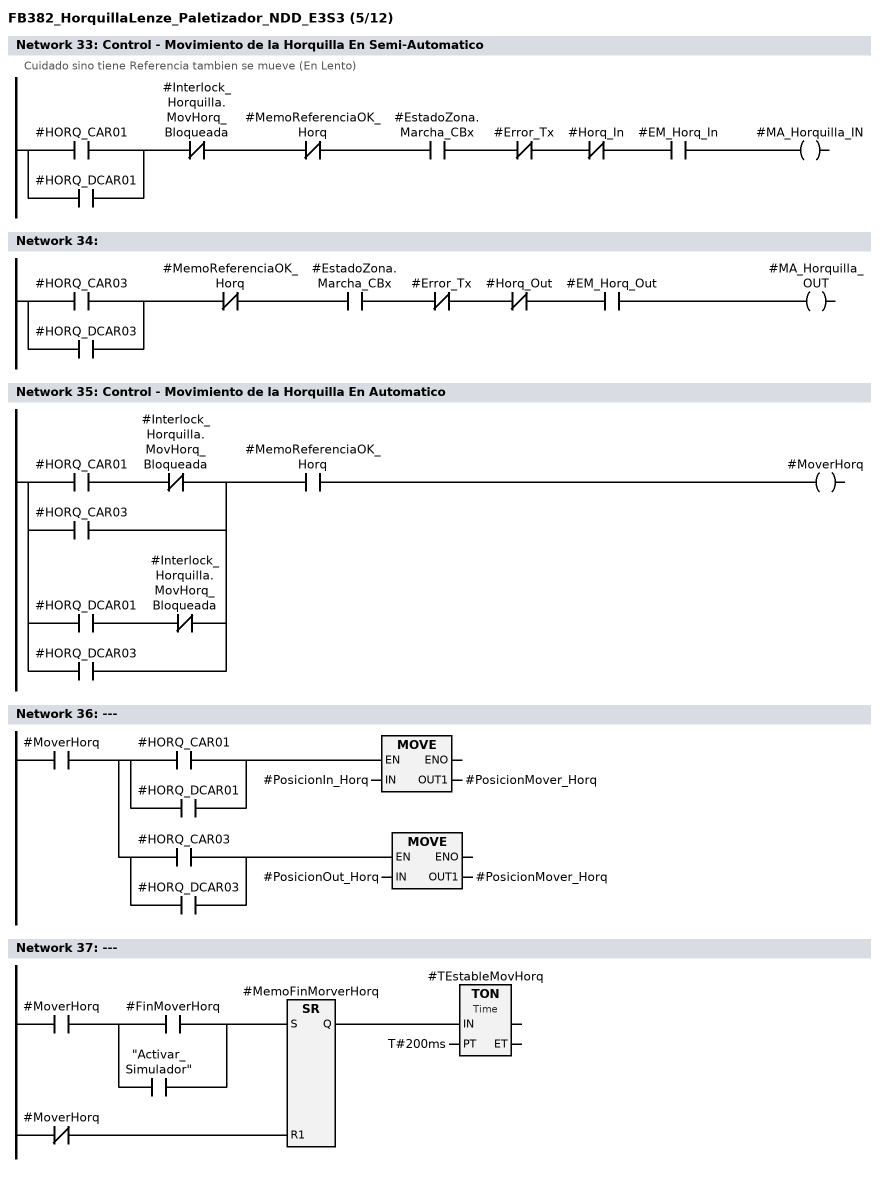
   RUNG wire#powerrail
      Contact( #HORQ_CAR01 )
      wire#w1
      I_Contact( #Interlock_Horquilla.MovHorq_Bloqueada )
      I_Contact( #MemoReferenciaOK_Horq )
      Contact( #EstadoZona.Marcha_CBx )
      I_Contact( #Error_Tx )
      I_Contact( #Horq_In )
      Contact( #EM_Horq_In )
      Coil( #MA_Horquilla_IN )
   END_RUNG
   RUNG wire#powerrail
      Contact( #HORQ_DCAR01 )
   END_RUNG wire#w1
   // the same network as SCL:
   #MA_Horquilla_IN := (#HORQ_CAR01 OR #HORQ_DCAR01) AND NOT #Interlock_Horquilla.MovHorq_Bloqueada AND NOT #MemoReferenciaOK_Horq AND #EstadoZona.Marcha_CBx AND NOT #Error_Tx AND NOT #Horq_In AND #EM_Horq_In;
END_REGION

REGION Network 34
   RUNG wire#powerrail
      Contact( #HORQ_CAR03 )
      wire#w1
      I_Contact( #MemoReferenciaOK_Horq )
      Contact( #EstadoZona.Marcha_CBx )
      I_Contact( #Error_Tx )
      I_Contact( #Horq_Out )
      Contact( #EM_Horq_Out )
      Coil( #MA_Horquilla_OUT )
   END_RUNG
   RUNG wire#powerrail
      Contact( #HORQ_DCAR03 )
   END_RUNG wire#w1
   // the same network as SCL:
   #MA_Horquilla_OUT := (#HORQ_CAR03 OR #HORQ_DCAR03) AND NOT #MemoReferenciaOK_Horq AND #EstadoZona.Marcha_CBx AND NOT #Error_Tx AND NOT #Horq_Out AND #EM_Horq_Out;
END_REGION

REGION Network 35: Control - Movimiento de la Horquilla En Automatico
   RUNG wire#powerrail
      Contact( #HORQ_CAR01 )
      I_Contact( #Interlock_Horquilla.MovHorq_Bloqueada )
      wire#w1
      Contact( #MemoReferenciaOK_Horq )
      Coil( #MoverHorq )
   END_RUNG
   RUNG wire#powerrail
      Contact( #HORQ_CAR03 )
   END_RUNG wire#w1
   RUNG wire#powerrail
      Contact( #HORQ_DCAR01 )
      I_Contact( #Interlock_Horquilla.MovHorq_Bloqueada )
   END_RUNG wire#w1
   RUNG wire#powerrail
      Contact( #HORQ_DCAR03 )
   END_RUNG wire#w1
   // the same network as SCL:
   #MoverHorq := ((#HORQ_CAR01 AND NOT #Interlock_Horquilla.MovHorq_Bloqueada) OR #HORQ_CAR03 OR (#HORQ_DCAR01 AND NOT #Interlock_Horquilla.MovHorq_Bloqueada) OR #HORQ_DCAR03) AND #MemoReferenciaOK_Horq;
END_REGION

REGION Network 36: ---
   RUNG wire#powerrail
      Contact( #MoverHorq )
      wire#w1
      Contact( #HORQ_CAR01 )
      wire#w2
      { S7_GenerateENO := "TRUE" } Move(in := #PosicionIn_Horq, out1 => #PosicionMover_Horq)
   END_RUNG
   RUNG wire#w1
      Contact( #HORQ_DCAR01 )
   END_RUNG wire#w2
   RUNG wire#w1
      Contact( #HORQ_CAR03 )
      wire#w3
      { S7_GenerateENO := "TRUE" } Move(in := #PosicionOut_Horq, out1 => #PosicionMover_Horq)
   END_RUNG
   RUNG wire#w1
      Contact( #HORQ_DCAR03 )
   END_RUNG wire#w3
   // the same network as SCL:
   IF #MoverHorq AND (#HORQ_CAR01 OR #HORQ_DCAR01) THEN #PosicionMover_Horq := #PosicionIn_Horq; END_IF;
   IF #MoverHorq AND (#HORQ_CAR03 OR #HORQ_DCAR03) THEN #PosicionMover_Horq := #PosicionOut_Horq; END_IF;
END_REGION

REGION Network 37: ---
   RUNG wire#powerrail
      Contact( #MoverHorq )
      wire#w1
      Contact( #FinMoverHorq )
      wire#w2
      S_SR(operand := #MemoFinMorverHorq, r1 := wire#w3)
      { S7_Templates := "time_type := Time" } #TEstableMovHorq.TON(pt := T#200ms, et =>)
   END_RUNG
   RUNG wire#w1
      Contact( "Activar_Simulador" )
   END_RUNG wire#w2
   RUNG wire#powerrail
      I_Contact( #MoverHorq )
   END_RUNG wire#w3
   // the same network as SCL:
   IF #MoverHorq AND (#FinMoverHorq OR "Activar_Simulador") THEN
       #MemoFinMorverHorq := TRUE;   // SR flip-flop
   END_IF;
   IF NOT #MoverHorq THEN #MemoFinMorverHorq := FALSE; END_IF;
   #TEstableMovHorq(IN := #MemoFinMorverHorq, PT := T#200ms);   // TON
END_REGION

REGION Network 38: Fisico - Movimiento de la Horquilla
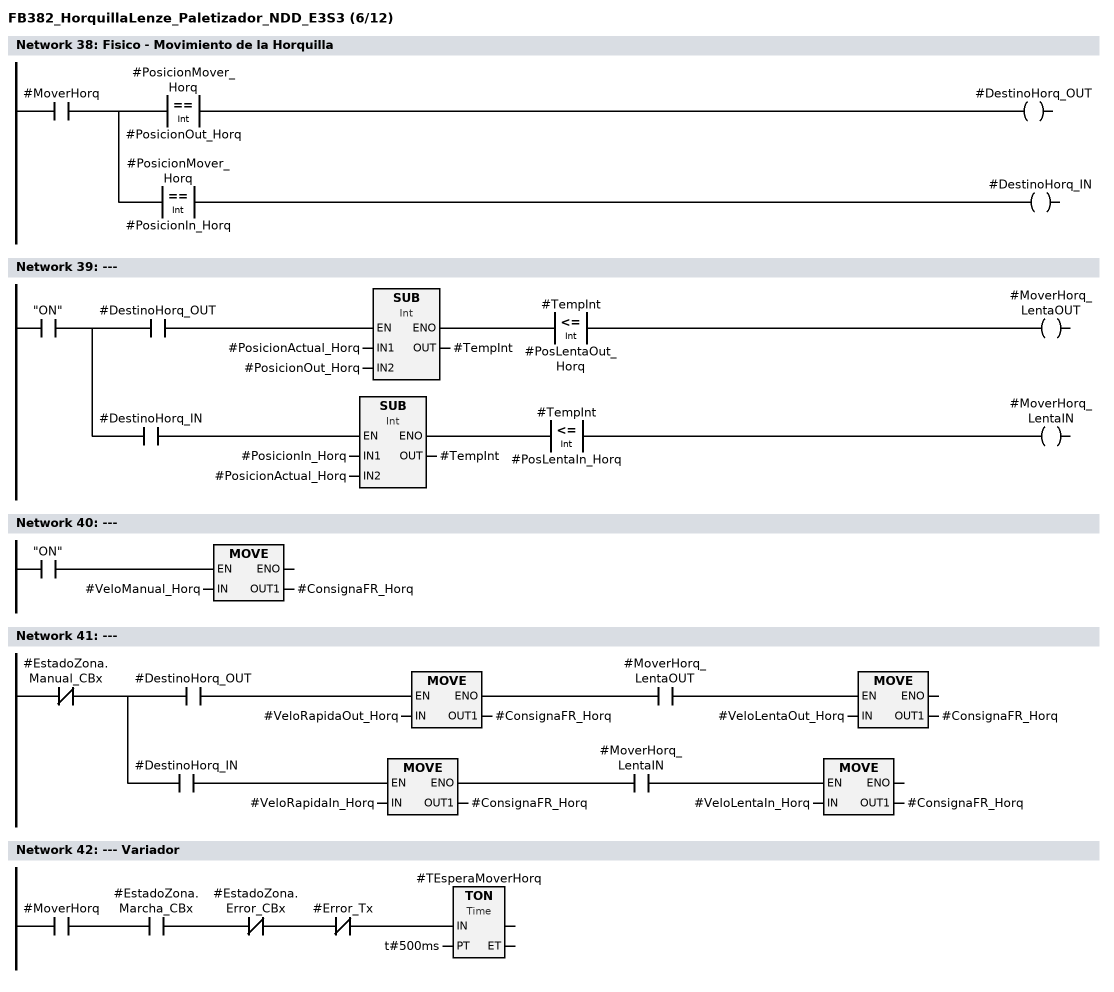
   RUNG wire#powerrail
      Contact( #MoverHorq )
      wire#w1
      { S7_Templates := "SrcType := Int" } EQ_Contact(in1 := #PosicionMover_Horq, in2 := #PosicionOut_Horq)
      Coil( #DestinoHorq_OUT )
   END_RUNG
   RUNG wire#w1
      { S7_Templates := "SrcType := Int" } EQ_Contact(in1 := #PosicionMover_Horq, in2 := #PosicionIn_Horq)
      Coil( #DestinoHorq_IN )
   END_RUNG
   // the same network as SCL:
   #DestinoHorq_OUT := #MoverHorq AND (#PosicionMover_Horq = #PosicionOut_Horq);
   #DestinoHorq_IN := #MoverHorq AND (#PosicionMover_Horq = #PosicionIn_Horq);
END_REGION

REGION Network 39: ---
   RUNG wire#powerrail
      Contact( "ON" )
      wire#w1
      Contact( #DestinoHorq_OUT )
      { S7_Templates := "SrcType := Int"; S7_GenerateENO := "TRUE" } Sub(in1 := #PosicionActual_Horq, in2 := #PosicionOut_Horq, out => #TempInt)
      { S7_Templates := "SrcType := Int" } LE_Contact(in1 := #TempInt, in2 := #PosLentaOut_Horq)
      Coil( #MoverHorq_LentaOUT )
   END_RUNG
   RUNG wire#w1
      Contact( #DestinoHorq_IN )
      { S7_Templates := "SrcType := Int"; S7_GenerateENO := "TRUE" } Sub(in1 := #PosicionIn_Horq, in2 := #PosicionActual_Horq, out => #TempInt)
      { S7_Templates := "SrcType := Int" } LE_Contact(in1 := #TempInt, in2 := #PosLentaIn_Horq)
      Coil( #MoverHorq_LentaIN )
   END_RUNG
   // the same network as SCL:
   // ENO of a box is taken as its EN; it also drops when the box reports an error
   #_w1 := "ON" AND #DestinoHorq_OUT;
   IF #_w1 THEN #TempInt := #PosicionActual_Horq - #PosicionOut_Horq; END_IF;
   #MoverHorq_LentaOUT := #_w1 AND (#TempInt <= #PosLentaOut_Horq);
   #_w2 := "ON" AND #DestinoHorq_IN;
   IF #_w2 THEN #TempInt := #PosicionIn_Horq - #PosicionActual_Horq; END_IF;
   #MoverHorq_LentaIN := #_w2 AND (#TempInt <= #PosLentaIn_Horq);
END_REGION

REGION Network 40: ---
   RUNG wire#powerrail
      Contact( "ON" )
      { S7_GenerateENO := "TRUE" } Move(in := #VeloManual_Horq, out1 => #ConsignaFR_Horq)
   END_RUNG
   // the same network as SCL:
   IF "ON" THEN #ConsignaFR_Horq := #VeloManual_Horq; END_IF;
END_REGION

REGION Network 41: ---
   RUNG wire#powerrail
      I_Contact( #EstadoZona.Manual_CBx )
      wire#w1
      Contact( #DestinoHorq_OUT )
      { S7_GenerateENO := "TRUE" } Move(in := #VeloRapidaOut_Horq, out1 => #ConsignaFR_Horq)
      Contact( #MoverHorq_LentaOUT )
      { S7_GenerateENO := "TRUE" } Move(in := #VeloLentaOut_Horq, out1 => #ConsignaFR_Horq)
   END_RUNG
   RUNG wire#w1
      Contact( #DestinoHorq_IN )
      { S7_GenerateENO := "TRUE" } Move(in := #VeloRapidaIn_Horq, out1 => #ConsignaFR_Horq)
      Contact( #MoverHorq_LentaIN )
      { S7_GenerateENO := "TRUE" } Move(in := #VeloLentaIn_Horq, out1 => #ConsignaFR_Horq)
   END_RUNG
   // the same network as SCL:
   // ENO of a box is taken as its EN; it also drops when the box reports an error
   #_w1 := NOT #EstadoZona.Manual_CBx;
   #_w2 := #_w1 AND #DestinoHorq_OUT;
   IF #_w2 THEN #ConsignaFR_Horq := #VeloRapidaOut_Horq; END_IF;
   IF #_w2 AND #MoverHorq_LentaOUT THEN #ConsignaFR_Horq := #VeloLentaOut_Horq; END_IF;
   #_w3 := #_w1 AND #DestinoHorq_IN;
   IF #_w3 THEN #ConsignaFR_Horq := #VeloRapidaIn_Horq; END_IF;
   IF #_w3 AND #MoverHorq_LentaIN THEN #ConsignaFR_Horq := #VeloLentaIn_Horq; END_IF;
END_REGION

REGION Network 42: --- Variador
   RUNG wire#powerrail
      Contact( #MoverHorq )
      Contact( #EstadoZona.Marcha_CBx )
      I_Contact( #EstadoZona.Error_CBx )
      I_Contact( #Error_Tx )
      { S7_Templates := "time_type := Time" } #TEsperaMoverHorq.TON(pt := t#500ms, et =>)
   END_RUNG
   // the same network as SCL:
   #TEsperaMoverHorq(IN := #MoverHorq AND #EstadoZona.Marcha_CBx AND NOT #EstadoZona.Error_CBx AND NOT #Error_Tx,   // TON
                     PT := t#500ms);
END_REGION

REGION Network 43: ----
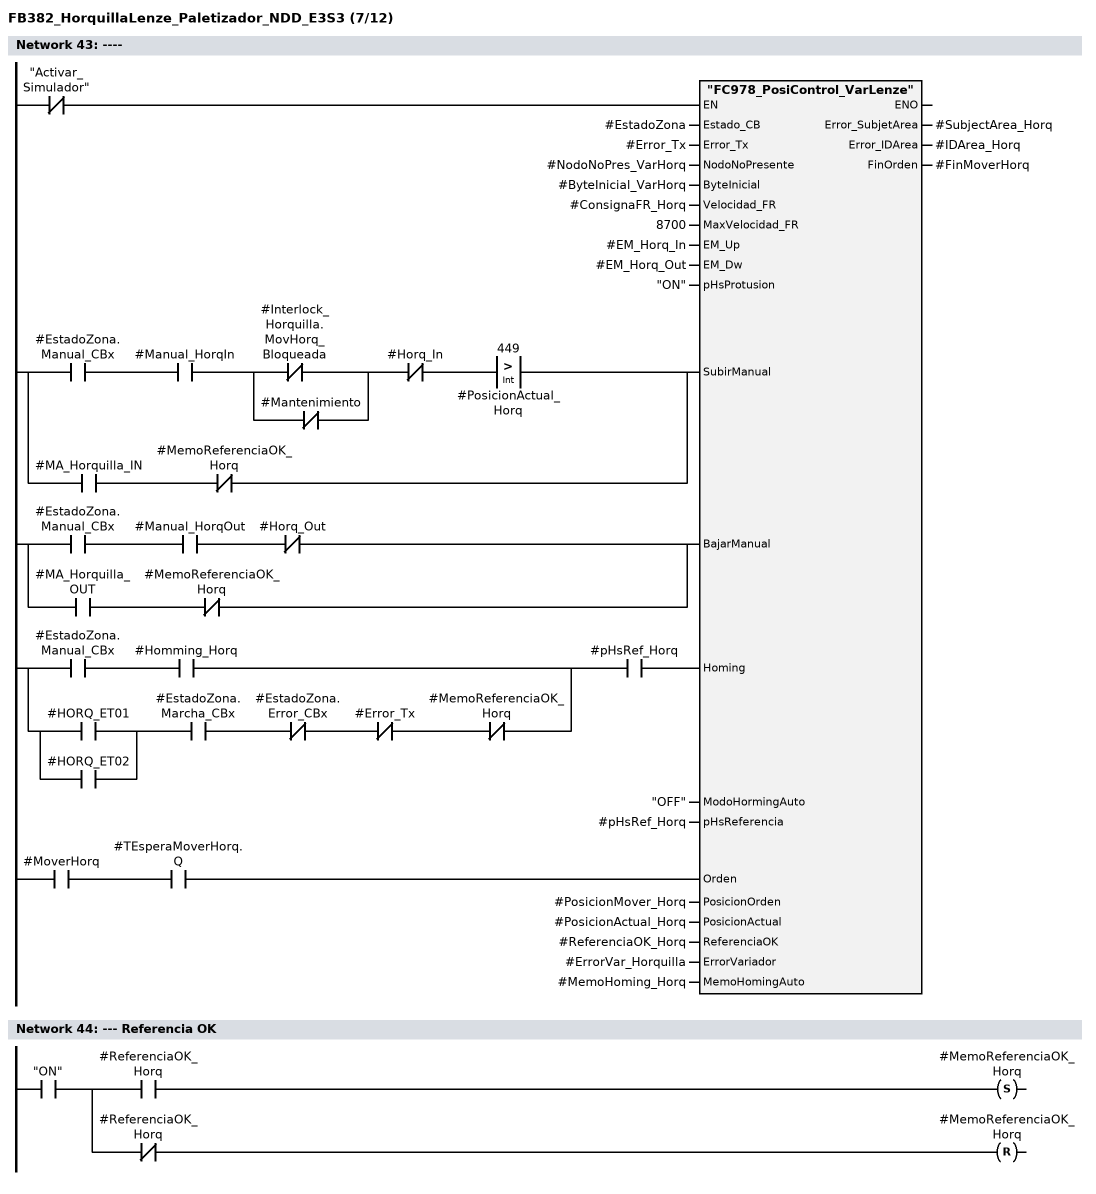
   RUNG wire#powerrail
      I_Contact( "Activar_Simulador" )
      "FC978_PosiControl_VarLenze"(SubirManual := wire#w3, BajarManual := wire#w4, Homing := wire#w7, Orden := wire#w8, Estado_CB := #EstadoZona, Error_Tx := #Error_Tx, NodoNoPresente := #NodoNoPres_VarHorq, ByteInicial := #ByteInicial_VarHorq, Velocidad_FR := #ConsignaFR_Horq, MaxVelocidad_FR := 8700, EM_Up := #EM_Horq_In, EM_Dw := #EM_Horq_Out, pHsProtusion := "ON", ModoHormingAuto := "OFF", pHsReferencia := #pHsRef_Horq, PosicionOrden := #PosicionMover_Horq, PosicionActual := #PosicionActual_Horq, ReferenciaOK := #ReferenciaOK_Horq, ErrorVariador := #ErrorVar_Horquilla, MemoHomingAuto := #MemoHoming_Horq, Error_SubjetArea => #SubjectArea_Horq, Error_IDArea => #IDArea_Horq, FinOrden => #FinMoverHorq)
   END_RUNG
   RUNG wire#powerrail
      Contact( #EstadoZona.Manual_CBx )
      Contact( #Manual_HorqIn )
      wire#w1
      I_Contact( #Interlock_Horquilla.MovHorq_Bloqueada )
      wire#w2
      I_Contact( #Horq_In )
      { S7_Templates := "SrcType := Int" } GT_Contact(in1 := 449, in2 := #PosicionActual_Horq)
   END_RUNG wire#w3
   RUNG wire#w1
      I_Contact( #Mantenimiento )
   END_RUNG wire#w2
   RUNG wire#powerrail
      Contact( #MA_Horquilla_IN )
      I_Contact( #MemoReferenciaOK_Horq )
   END_RUNG wire#w3
   RUNG wire#powerrail
      Contact( #EstadoZona.Manual_CBx )
      Contact( #Manual_HorqOut )
      I_Contact( #Horq_Out )
   END_RUNG wire#w4
   RUNG wire#powerrail
      Contact( #MA_Horquilla_OUT )
      I_Contact( #MemoReferenciaOK_Horq )
   END_RUNG wire#w4
   RUNG wire#powerrail
      Contact( #EstadoZona.Manual_CBx )
      Contact( #Homming_Horq )
      wire#w5
      Contact( #pHsRef_Horq )
   END_RUNG wire#w7
   RUNG wire#powerrail
      Contact( #HORQ_ET01 )
      wire#w6
      Contact( #EstadoZona.Marcha_CBx )
      I_Contact( #EstadoZona.Error_CBx )
      I_Contact( #Error_Tx )
      I_Contact( #MemoReferenciaOK_Horq )
   END_RUNG wire#w5
   RUNG wire#powerrail
      Contact( #HORQ_ET02 )
   END_RUNG wire#w6
   RUNG wire#powerrail
      Contact( #MoverHorq )
      Contact( #TEsperaMoverHorq.Q )
   END_RUNG wire#w8
   // the same network as SCL:
   IF NOT "Activar_Simulador" THEN
       "FC978_PosiControl_VarLenze"(Estado_CB := #EstadoZona,
                               Error_Tx := #Error_Tx,
                               NodoNoPresente := #NodoNoPres_VarHorq,
                               ByteInicial := #ByteInicial_VarHorq,
                               Velocidad_FR := #ConsignaFR_Horq,
                               MaxVelocidad_FR := 8700,
                               EM_Up := #EM_Horq_In,
                               EM_Dw := #EM_Horq_Out,
                               pHsProtusion := "ON",
                               SubirManual := (#EstadoZona.Manual_CBx AND #Manual_HorqIn AND (NOT #Interlock_Horquilla.MovHorq_Bloqueada OR NOT #Mantenimiento) AND NOT #Horq_In AND (449 > #PosicionActual_Horq)) OR (#MA_Horquilla_IN AND NOT #MemoReferenciaOK_Horq),
                               BajarManual := (#EstadoZona.Manual_CBx AND #Manual_HorqOut AND NOT #Horq_Out) OR (#MA_Horquilla_OUT AND NOT #MemoReferenciaOK_Horq),
                               Homing := ((#EstadoZona.Manual_CBx AND #Homming_Horq) OR ((#HORQ_ET01 OR #HORQ_ET02) AND #EstadoZona.Marcha_CBx AND NOT #EstadoZona.Error_CBx AND NOT #Error_Tx AND NOT #MemoReferenciaOK_Horq)) AND #pHsRef_Horq,
                               ModoHormingAuto := "OFF",
                               pHsReferencia := #pHsRef_Horq,
                               Orden := #MoverHorq AND #TEsperaMoverHorq.Q,
                               PosicionOrden := #PosicionMover_Horq,
                               PosicionActual := #PosicionActual_Horq,
                               ReferenciaOK := #ReferenciaOK_Horq,
                               ErrorVariador := #ErrorVar_Horquilla,
                               MemoHomingAuto := #MemoHoming_Horq,
                               Error_SubjetArea => #SubjectArea_Horq,
                               Error_IDArea => #IDArea_Horq,
                               FinOrden => #FinMoverHorq);
   END_IF;
END_REGION

REGION Network 44: --- Referencia OK
   RUNG wire#powerrail
      Contact( "ON" )
      wire#w1
      Contact( #ReferenciaOK_Horq )
      S_Coil( #MemoReferenciaOK_Horq )
   END_RUNG
   RUNG wire#w1
      I_Contact( #ReferenciaOK_Horq )
      R_Coil( #MemoReferenciaOK_Horq )
   END_RUNG
   // the same network as SCL:
   IF "ON" AND #ReferenciaOK_Horq THEN #MemoReferenciaOK_Horq := TRUE; END_IF;
   IF "ON" AND NOT #ReferenciaOK_Horq THEN #MemoReferenciaOK_Horq := FALSE; END_IF;
END_REGION

REGION Network 45: Errores de la Horquilla
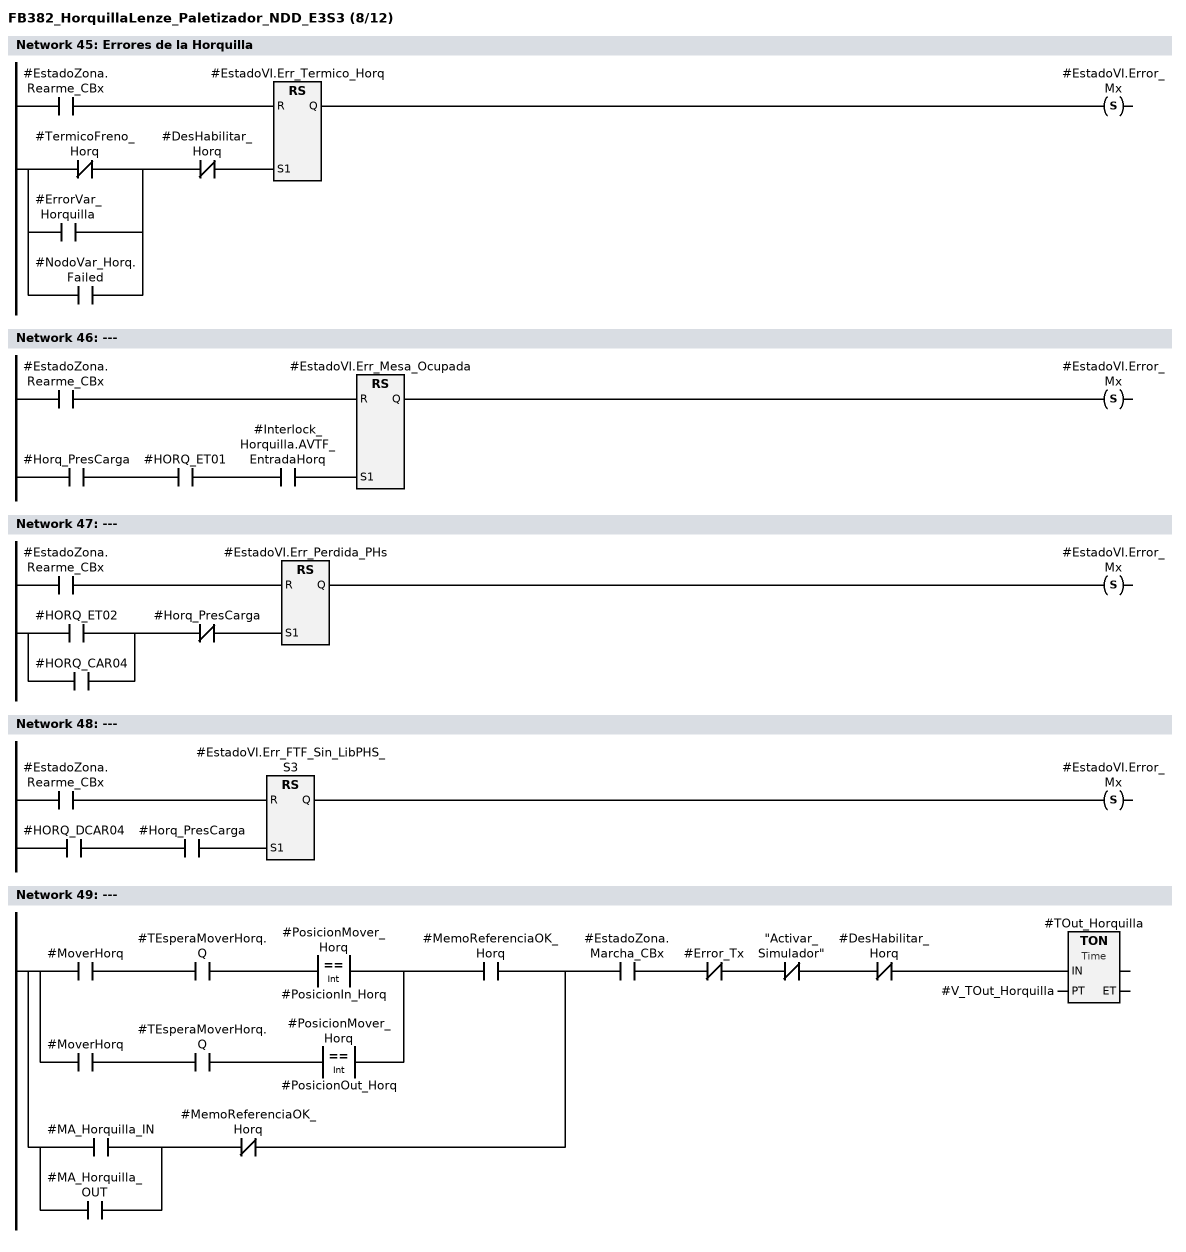
   RUNG wire#powerrail
      Contact( #EstadoZona.Rearme_CBx )
      S_RS(operand := #EstadoVI.Err_Termico_Horq, s1 := wire#w2)
      S_Coil( #EstadoVI.Error_Mx )
   END_RUNG
   RUNG wire#powerrail
      I_Contact( #TermicoFreno_Horq )
      wire#w1
      I_Contact( #DesHabilitar_Horq )
   END_RUNG wire#w2
   RUNG wire#powerrail
      Contact( #ErrorVar_Horquilla )
   END_RUNG wire#w1
   RUNG wire#powerrail
      Contact( #NodoVar_Horq.Failed )
   END_RUNG wire#w1
   // the same network as SCL:
   IF #EstadoZona.Rearme_CBx THEN
       #EstadoVI.Err_Termico_Horq := FALSE;   // RS flip-flop
   END_IF;
   IF (NOT #TermicoFreno_Horq OR #ErrorVar_Horquilla OR #NodoVar_Horq.Failed) AND NOT #DesHabilitar_Horq THEN
       #EstadoVI.Err_Termico_Horq := TRUE;
   END_IF;
   IF #EstadoVI.Err_Termico_Horq THEN #EstadoVI.Error_Mx := TRUE; END_IF;
END_REGION

REGION Network 46: ---
   RUNG wire#powerrail
      Contact( #EstadoZona.Rearme_CBx )
      S_RS(operand := #EstadoVI.Err_Mesa_Ocupada, s1 := wire#w1)
      S_Coil( #EstadoVI.Error_Mx )
   END_RUNG
   RUNG wire#powerrail
      Contact( #Horq_PresCarga )
      Contact( #HORQ_ET01 )
      Contact( #Interlock_Horquilla.AVTF_EntradaHorq )
   END_RUNG wire#w1
   // the same network as SCL:
   IF #EstadoZona.Rearme_CBx THEN
       #EstadoVI.Err_Mesa_Ocupada := FALSE;   // RS flip-flop
   END_IF;
   IF #Horq_PresCarga AND #HORQ_ET01 AND #Interlock_Horquilla.AVTF_EntradaHorq THEN
       #EstadoVI.Err_Mesa_Ocupada := TRUE;
   END_IF;
   IF #EstadoVI.Err_Mesa_Ocupada THEN #EstadoVI.Error_Mx := TRUE; END_IF;
END_REGION

REGION Network 47: ---
   RUNG wire#powerrail
      Contact( #EstadoZona.Rearme_CBx )
      S_RS(operand := #EstadoVI.Err_Perdida_PHs, s1 := wire#w2)
      S_Coil( #EstadoVI.Error_Mx )
   END_RUNG
   RUNG wire#powerrail
      Contact( #HORQ_ET02 )
      wire#w1
      I_Contact( #Horq_PresCarga )
   END_RUNG wire#w2
   RUNG wire#powerrail
      Contact( #HORQ_CAR04 )
   END_RUNG wire#w1
   // the same network as SCL:
   IF #EstadoZona.Rearme_CBx THEN
       #EstadoVI.Err_Perdida_PHs := FALSE;   // RS flip-flop
   END_IF;
   IF (#HORQ_ET02 OR #HORQ_CAR04) AND NOT #Horq_PresCarga THEN #EstadoVI.Err_Perdida_PHs := TRUE; END_IF;
   IF #EstadoVI.Err_Perdida_PHs THEN #EstadoVI.Error_Mx := TRUE; END_IF;
END_REGION

REGION Network 48: ---
   RUNG wire#powerrail
      Contact( #EstadoZona.Rearme_CBx )
      S_RS(operand := #EstadoVI.Err_FTF_Sin_LibPHS_S3, s1 := wire#w1)
      S_Coil( #EstadoVI.Error_Mx )
   END_RUNG
   RUNG wire#powerrail
      Contact( #HORQ_DCAR04 )
      Contact( #Horq_PresCarga )
   END_RUNG wire#w1
   // the same network as SCL:
   IF #EstadoZona.Rearme_CBx THEN
       #EstadoVI.Err_FTF_Sin_LibPHS_S3 := FALSE;   // RS flip-flop
   END_IF;
   IF #HORQ_DCAR04 AND #Horq_PresCarga THEN #EstadoVI.Err_FTF_Sin_LibPHS_S3 := TRUE; END_IF;
   IF #EstadoVI.Err_FTF_Sin_LibPHS_S3 THEN #EstadoVI.Error_Mx := TRUE; END_IF;
END_REGION

REGION Network 49: ---
   RUNG wire#powerrail
      Contact( #MoverHorq )
      Contact( #TEsperaMoverHorq.Q )
      { S7_Templates := "SrcType := Int" } EQ_Contact(in1 := #PosicionMover_Horq, in2 := #PosicionIn_Horq)
      wire#w1
      Contact( #MemoReferenciaOK_Horq )
      wire#w2
      Contact( #EstadoZona.Marcha_CBx )
      I_Contact( #Error_Tx )
      I_Contact( "Activar_Simulador" )
      I_Contact( #DesHabilitar_Horq )
      { S7_Templates := "time_type := Time" } #TOut_Horquilla.TON(pt := #V_TOut_Horquilla, et =>)
   END_RUNG
   RUNG wire#powerrail
      Contact( #MoverHorq )
      Contact( #TEsperaMoverHorq.Q )
      { S7_Templates := "SrcType := Int" } EQ_Contact(in1 := #PosicionMover_Horq, in2 := #PosicionOut_Horq)
   END_RUNG wire#w1
   RUNG wire#powerrail
      Contact( #MA_Horquilla_IN )
      wire#w3
      I_Contact( #MemoReferenciaOK_Horq )
   END_RUNG wire#w2
   RUNG wire#powerrail
      Contact( #MA_Horquilla_OUT )
   END_RUNG wire#w3
   // the same network as SCL:
   #TOut_Horquilla(IN := ((((#MoverHorq AND #TEsperaMoverHorq.Q AND (#PosicionMover_Horq = #PosicionIn_Horq)) OR (#MoverHorq AND #TEsperaMoverHorq.Q AND (#PosicionMover_Horq = #PosicionOut_Horq))) AND #MemoReferenciaOK_Horq) OR ((#MA_Horquilla_IN OR #MA_Horquilla_OUT) AND NOT #MemoReferenciaOK_Horq)) AND #EstadoZona.Marcha_CBx AND NOT #Error_Tx AND NOT "Activar_Simulador" AND NOT #DesHabilitar_Horq,   // TON
                   PT := #V_TOut_Horquilla);
END_REGION

REGION Network 50: ---
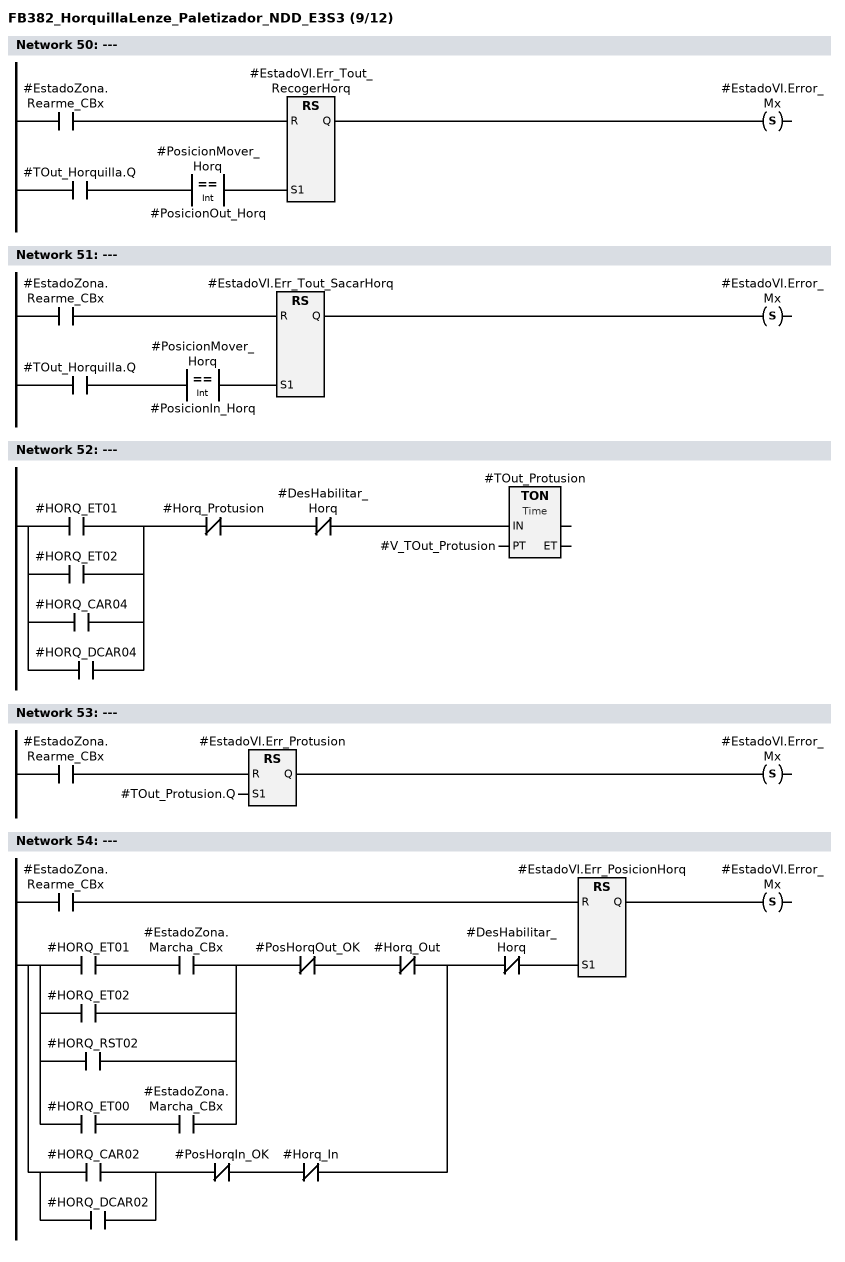
   RUNG wire#powerrail
      Contact( #EstadoZona.Rearme_CBx )
      S_RS(operand := #EstadoVI.Err_Tout_RecogerHorq, s1 := wire#w1)
      S_Coil( #EstadoVI.Error_Mx )
   END_RUNG
   RUNG wire#powerrail
      Contact( #TOut_Horquilla.Q )
      { S7_Templates := "SrcType := Int" } EQ_Contact(in1 := #PosicionMover_Horq, in2 := #PosicionOut_Horq)
   END_RUNG wire#w1
   // the same network as SCL:
   IF #EstadoZona.Rearme_CBx THEN
       #EstadoVI.Err_Tout_RecogerHorq := FALSE;   // RS flip-flop
   END_IF;
   IF #TOut_Horquilla.Q AND (#PosicionMover_Horq = #PosicionOut_Horq) THEN
       #EstadoVI.Err_Tout_RecogerHorq := TRUE;
   END_IF;
   IF #EstadoVI.Err_Tout_RecogerHorq THEN #EstadoVI.Error_Mx := TRUE; END_IF;
END_REGION

REGION Network 51: ---
   RUNG wire#powerrail
      Contact( #EstadoZona.Rearme_CBx )
      S_RS(operand := #EstadoVI.Err_Tout_SacarHorq, s1 := wire#w1)
      S_Coil( #EstadoVI.Error_Mx )
   END_RUNG
   RUNG wire#powerrail
      Contact( #TOut_Horquilla.Q )
      { S7_Templates := "SrcType := Int" } EQ_Contact(in1 := #PosicionMover_Horq, in2 := #PosicionIn_Horq)
   END_RUNG wire#w1
   // the same network as SCL:
   IF #EstadoZona.Rearme_CBx THEN
       #EstadoVI.Err_Tout_SacarHorq := FALSE;   // RS flip-flop
   END_IF;
   IF #TOut_Horquilla.Q AND (#PosicionMover_Horq = #PosicionIn_Horq) THEN
       #EstadoVI.Err_Tout_SacarHorq := TRUE;
   END_IF;
   IF #EstadoVI.Err_Tout_SacarHorq THEN #EstadoVI.Error_Mx := TRUE; END_IF;
END_REGION

REGION Network 52: ---
   RUNG wire#powerrail
      Contact( #HORQ_ET01 )
      wire#w1
      I_Contact( #Horq_Protusion )
      I_Contact( #DesHabilitar_Horq )
      { S7_Templates := "time_type := Time" } #TOut_Protusion.TON(pt := #V_TOut_Protusion, et =>)
   END_RUNG
   RUNG wire#powerrail
      Contact( #HORQ_ET02 )
   END_RUNG wire#w1
   RUNG wire#powerrail
      Contact( #HORQ_CAR04 )
   END_RUNG wire#w1
   RUNG wire#powerrail
      Contact( #HORQ_DCAR04 )
   END_RUNG wire#w1
   // the same network as SCL:
   #TOut_Protusion(IN := (#HORQ_ET01 OR #HORQ_ET02 OR #HORQ_CAR04 OR #HORQ_DCAR04) AND NOT #Horq_Protusion AND NOT #DesHabilitar_Horq,   // TON
                   PT := #V_TOut_Protusion);
END_REGION

REGION Network 53: ---
   RUNG wire#powerrail
      Contact( #EstadoZona.Rearme_CBx )
      S_RS(operand := #EstadoVI.Err_Protusion, s1 := #TOut_Protusion.Q)
      S_Coil( #EstadoVI.Error_Mx )
   END_RUNG
   // the same network as SCL:
   IF #EstadoZona.Rearme_CBx THEN
       #EstadoVI.Err_Protusion := FALSE;   // RS flip-flop
   END_IF;
   IF #TOut_Protusion.Q THEN #EstadoVI.Err_Protusion := TRUE; END_IF;
   IF #EstadoVI.Err_Protusion THEN #EstadoVI.Error_Mx := TRUE; END_IF;
END_REGION

REGION Network 54: ---
   RUNG wire#powerrail
      Contact( #EstadoZona.Rearme_CBx )
      S_RS(operand := #EstadoVI.Err_PosicionHorq, s1 := wire#w4)
      S_Coil( #EstadoVI.Error_Mx )
   END_RUNG
   RUNG wire#powerrail
      Contact( #HORQ_ET01 )
      Contact( #EstadoZona.Marcha_CBx )
      wire#w1
      I_Contact( #PosHorqOut_OK )
      I_Contact( #Horq_Out )
      wire#w2
      I_Contact( #DesHabilitar_Horq )
   END_RUNG wire#w4
   RUNG wire#powerrail
      Contact( #HORQ_ET02 )
   END_RUNG wire#w1
   RUNG wire#powerrail
      Contact( #HORQ_RST02 )
   END_RUNG wire#w1
   RUNG wire#powerrail
      Contact( #HORQ_ET00 )
      Contact( #EstadoZona.Marcha_CBx )
   END_RUNG wire#w1
   RUNG wire#powerrail
      Contact( #HORQ_CAR02 )
      wire#w3
      I_Contact( #PosHorqIn_OK )
      I_Contact( #Horq_In )
   END_RUNG wire#w2
   RUNG wire#powerrail
      Contact( #HORQ_DCAR02 )
   END_RUNG wire#w3
   // the same network as SCL:
   IF #EstadoZona.Rearme_CBx THEN
       #EstadoVI.Err_PosicionHorq := FALSE;   // RS flip-flop
   END_IF;
   IF ((((#HORQ_ET01 AND #EstadoZona.Marcha_CBx) OR #HORQ_ET02 OR #HORQ_RST02 OR (#HORQ_ET00 AND #EstadoZona.Marcha_CBx)) AND NOT #PosHorqOut_OK AND NOT #Horq_Out) OR ((#HORQ_CAR02 OR #HORQ_DCAR02) AND NOT #PosHorqIn_OK AND NOT #Horq_In)) AND NOT #DesHabilitar_Horq THEN
       #EstadoVI.Err_PosicionHorq := TRUE;
   END_IF;
   IF #EstadoVI.Err_PosicionHorq THEN #EstadoVI.Error_Mx := TRUE; END_IF;
END_REGION

REGION Network 55: ----
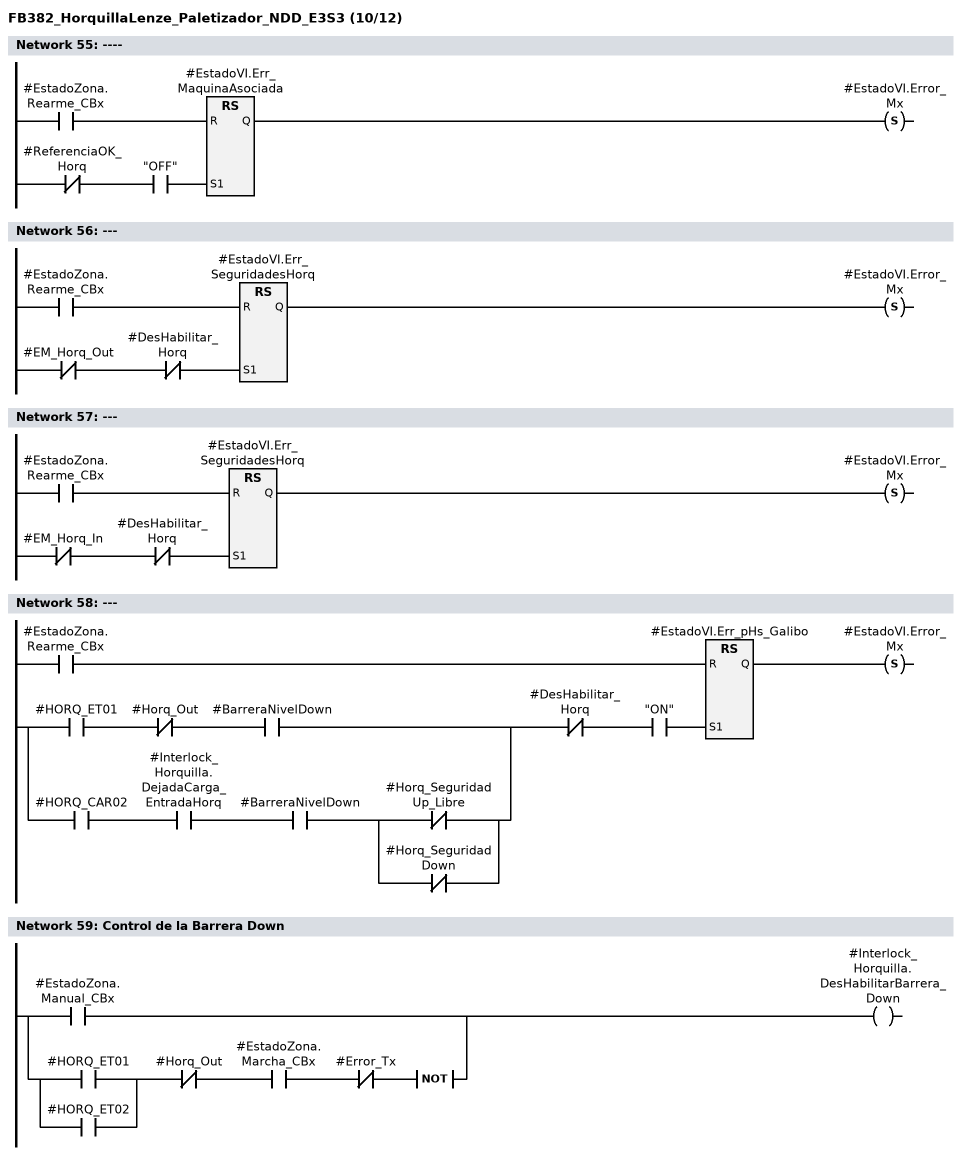
   RUNG wire#powerrail
      Contact( #EstadoZona.Rearme_CBx )
      S_RS(operand := #EstadoVI.Err_MaquinaAsociada, s1 := wire#w1)
      S_Coil( #EstadoVI.Error_Mx )
   END_RUNG
   RUNG wire#powerrail
      I_Contact( #ReferenciaOK_Horq )
      Contact( "OFF" )
   END_RUNG wire#w1
   // the same network as SCL:
   IF #EstadoZona.Rearme_CBx THEN
       #EstadoVI.Err_MaquinaAsociada := FALSE;   // RS flip-flop
   END_IF;
   IF NOT #ReferenciaOK_Horq AND "OFF" THEN #EstadoVI.Err_MaquinaAsociada := TRUE; END_IF;
   IF #EstadoVI.Err_MaquinaAsociada THEN #EstadoVI.Error_Mx := TRUE; END_IF;
END_REGION

REGION Network 56: ---
   RUNG wire#powerrail
      Contact( #EstadoZona.Rearme_CBx )
      S_RS(operand := #EstadoVI.Err_SeguridadesHorq, s1 := wire#w1)
      S_Coil( #EstadoVI.Error_Mx )
   END_RUNG
   RUNG wire#powerrail
      I_Contact( #EM_Horq_Out )
      I_Contact( #DesHabilitar_Horq )
   END_RUNG wire#w1
   // the same network as SCL:
   IF #EstadoZona.Rearme_CBx THEN
       #EstadoVI.Err_SeguridadesHorq := FALSE;   // RS flip-flop
   END_IF;
   IF NOT #EM_Horq_Out AND NOT #DesHabilitar_Horq THEN #EstadoVI.Err_SeguridadesHorq := TRUE; END_IF;
   IF #EstadoVI.Err_SeguridadesHorq THEN #EstadoVI.Error_Mx := TRUE; END_IF;
END_REGION

REGION Network 57: ---
   RUNG wire#powerrail
      Contact( #EstadoZona.Rearme_CBx )
      S_RS(operand := #EstadoVI.Err_SeguridadesHorq, s1 := wire#w1)
      S_Coil( #EstadoVI.Error_Mx )
   END_RUNG
   RUNG wire#powerrail
      I_Contact( #EM_Horq_In )
      I_Contact( #DesHabilitar_Horq )
   END_RUNG wire#w1
   // the same network as SCL:
   IF #EstadoZona.Rearme_CBx THEN
       #EstadoVI.Err_SeguridadesHorq := FALSE;   // RS flip-flop
   END_IF;
   IF NOT #EM_Horq_In AND NOT #DesHabilitar_Horq THEN #EstadoVI.Err_SeguridadesHorq := TRUE; END_IF;
   IF #EstadoVI.Err_SeguridadesHorq THEN #EstadoVI.Error_Mx := TRUE; END_IF;
END_REGION

REGION Network 58: ---
   RUNG wire#powerrail
      Contact( #EstadoZona.Rearme_CBx )
      S_RS(operand := #EstadoVI.Err_pHs_Galibo, s1 := wire#w3)
      S_Coil( #EstadoVI.Error_Mx )
   END_RUNG
   RUNG wire#powerrail
      Contact( #HORQ_ET01 )
      I_Contact( #Horq_Out )
      Contact( #BarreraNivelDown )
      wire#w1
      I_Contact( #DesHabilitar_Horq )
      Contact( "ON" )
   END_RUNG wire#w3
   RUNG wire#powerrail
      Contact( #HORQ_CAR02 )
      Contact( #Interlock_Horquilla.DejadaCarga_EntradaHorq )
      Contact( #BarreraNivelDown )
      wire#w2
      I_Contact( #Horq_SeguridadUp_Libre )
   END_RUNG wire#w1
   RUNG wire#w2
      I_Contact( #Horq_SeguridadDown )
   END_RUNG wire#w1
   // the same network as SCL:
   IF #EstadoZona.Rearme_CBx THEN
       #EstadoVI.Err_pHs_Galibo := FALSE;   // RS flip-flop
   END_IF;
   IF ((#HORQ_ET01 AND NOT #Horq_Out AND #BarreraNivelDown) OR (#HORQ_CAR02 AND #Interlock_Horquilla.DejadaCarga_EntradaHorq AND #BarreraNivelDown AND (NOT #Horq_SeguridadUp_Libre OR NOT #Horq_SeguridadDown))) AND NOT #DesHabilitar_Horq AND "ON" THEN
       #EstadoVI.Err_pHs_Galibo := TRUE;
   END_IF;
   IF #EstadoVI.Err_pHs_Galibo THEN #EstadoVI.Error_Mx := TRUE; END_IF;
END_REGION

REGION Network 59: Control de la Barrera Down
   RUNG wire#powerrail
      Contact( #EstadoZona.Manual_CBx )
      wire#w1
      Coil( #Interlock_Horquilla.DesHabilitarBarrera_Down )
   END_RUNG
   RUNG wire#powerrail
      Contact( #HORQ_ET01 )
      wire#w2
      I_Contact( #Horq_Out )
      Contact( #EstadoZona.Marcha_CBx )
      I_Contact( #Error_Tx )
      Not()
   END_RUNG wire#w1
   RUNG wire#powerrail
      Contact( #HORQ_ET02 )
   END_RUNG wire#w2
   // the same network as SCL:
   #Interlock_Horquilla.DesHabilitarBarrera_Down := #EstadoZona.Manual_CBx OR NOT ((#HORQ_ET01 OR #HORQ_ET02) AND NOT #Horq_Out AND #EstadoZona.Marcha_CBx AND NOT #Error_Tx);
END_REGION

REGION Network 60: Estados de la Horquilla
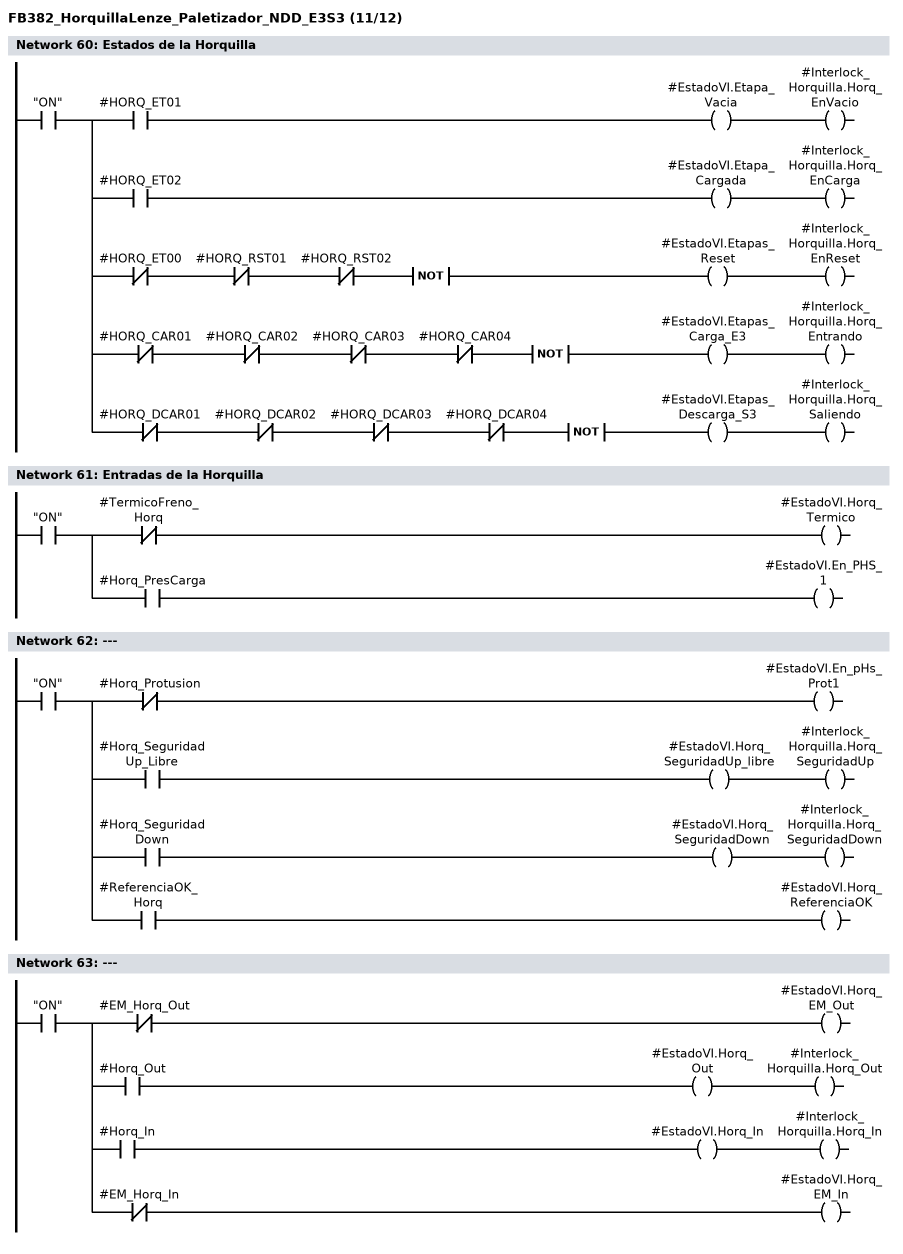
   RUNG wire#powerrail
      Contact( "ON" )
      wire#w1
      Contact( #HORQ_ET01 )
      Coil( #EstadoVI.Etapa_Vacia )
      Coil( #Interlock_Horquilla.Horq_EnVacio )
   END_RUNG
   RUNG wire#w1
      Contact( #HORQ_ET02 )
      Coil( #EstadoVI.Etapa_Cargada )
      Coil( #Interlock_Horquilla.Horq_EnCarga )
   END_RUNG
   RUNG wire#w1
      I_Contact( #HORQ_ET00 )
      I_Contact( #HORQ_RST01 )
      I_Contact( #HORQ_RST02 )
      Not()
      Coil( #EstadoVI.Etapas_Reset )
      Coil( #Interlock_Horquilla.Horq_EnReset )
   END_RUNG
   RUNG wire#w1
      I_Contact( #HORQ_CAR01 )
      I_Contact( #HORQ_CAR02 )
      I_Contact( #HORQ_CAR03 )
      I_Contact( #HORQ_CAR04 )
      Not()
      Coil( #EstadoVI.Etapas_Carga_E3 )
      Coil( #Interlock_Horquilla.Horq_Entrando )
   END_RUNG
   RUNG wire#w1
      I_Contact( #HORQ_DCAR01 )
      I_Contact( #HORQ_DCAR02 )
      I_Contact( #HORQ_DCAR03 )
      I_Contact( #HORQ_DCAR04 )
      Not()
      Coil( #EstadoVI.Etapas_Descarga_S3 )
      Coil( #Interlock_Horquilla.Horq_Saliendo )
   END_RUNG
   // the same network as SCL:
   #EstadoVI.Etapa_Vacia := "ON" AND #HORQ_ET01;
   #Interlock_Horquilla.Horq_EnVacio := #EstadoVI.Etapa_Vacia;
   #EstadoVI.Etapa_Cargada := "ON" AND #HORQ_ET02;
   #Interlock_Horquilla.Horq_EnCarga := #EstadoVI.Etapa_Cargada;
   #EstadoVI.Etapas_Reset := NOT ("ON" AND NOT #HORQ_ET00 AND NOT #HORQ_RST01 AND NOT #HORQ_RST02);
   #Interlock_Horquilla.Horq_EnReset := #EstadoVI.Etapas_Reset;
   #EstadoVI.Etapas_Carga_E3 := NOT ("ON" AND NOT #HORQ_CAR01 AND NOT #HORQ_CAR02 AND NOT #HORQ_CAR03 AND NOT #HORQ_CAR04);
   #Interlock_Horquilla.Horq_Entrando := #EstadoVI.Etapas_Carga_E3;
   #EstadoVI.Etapas_Descarga_S3 := NOT ("ON" AND NOT #HORQ_DCAR01 AND NOT #HORQ_DCAR02 AND NOT #HORQ_DCAR03 AND NOT #HORQ_DCAR04);
   #Interlock_Horquilla.Horq_Saliendo := #EstadoVI.Etapas_Descarga_S3;
END_REGION

REGION Network 61: Entradas de la Horquilla
   RUNG wire#powerrail
      Contact( "ON" )
      wire#w1
      I_Contact( #TermicoFreno_Horq )
      Coil( #EstadoVI.Horq_Termico )
   END_RUNG
   RUNG wire#w1
      Contact( #Horq_PresCarga )
      Coil( #EstadoVI.En_PHS_1 )
   END_RUNG
   // the same network as SCL:
   #EstadoVI.Horq_Termico := "ON" AND NOT #TermicoFreno_Horq;
   #EstadoVI.En_PHS_1 := "ON" AND #Horq_PresCarga;
END_REGION

REGION Network 62: ---
   RUNG wire#powerrail
      Contact( "ON" )
      wire#w1
      I_Contact( #Horq_Protusion )
      Coil( #EstadoVI.En_pHs_Prot1 )
   END_RUNG
   RUNG wire#w1
      Contact( #Horq_SeguridadUp_Libre )
      Coil( #EstadoVI.Horq_SeguridadUp_libre )
      Coil( #Interlock_Horquilla.Horq_SeguridadUp )
   END_RUNG
   RUNG wire#w1
      Contact( #Horq_SeguridadDown )
      Coil( #EstadoVI.Horq_SeguridadDown )
      Coil( #Interlock_Horquilla.Horq_SeguridadDown )
   END_RUNG
   RUNG wire#w1
      Contact( #ReferenciaOK_Horq )
      Coil( #EstadoVI.Horq_ReferenciaOK )
   END_RUNG
   // the same network as SCL:
   #EstadoVI.En_pHs_Prot1 := "ON" AND NOT #Horq_Protusion;
   #EstadoVI.Horq_SeguridadUp_libre := "ON" AND #Horq_SeguridadUp_Libre;
   #Interlock_Horquilla.Horq_SeguridadUp := #EstadoVI.Horq_SeguridadUp_libre;
   #EstadoVI.Horq_SeguridadDown := "ON" AND #Horq_SeguridadDown;
   #Interlock_Horquilla.Horq_SeguridadDown := #EstadoVI.Horq_SeguridadDown;
   #EstadoVI.Horq_ReferenciaOK := "ON" AND #ReferenciaOK_Horq;
END_REGION

REGION Network 63: ---
   RUNG wire#powerrail
      Contact( "ON" )
      wire#w1
      I_Contact( #EM_Horq_Out )
      Coil( #EstadoVI.Horq_EM_Out )
   END_RUNG
   RUNG wire#w1
      Contact( #Horq_Out )
      Coil( #EstadoVI.Horq_Out )
      Coil( #Interlock_Horquilla.Horq_Out )
   END_RUNG
   RUNG wire#w1
      Contact( #Horq_In )
      Coil( #EstadoVI.Horq_In )
      Coil( #Interlock_Horquilla.Horq_In )
   END_RUNG
   RUNG wire#w1
      I_Contact( #EM_Horq_In )
      Coil( #EstadoVI.Horq_EM_In )
   END_RUNG
   // the same network as SCL:
   #EstadoVI.Horq_EM_Out := "ON" AND NOT #EM_Horq_Out;
   #EstadoVI.Horq_Out := "ON" AND #Horq_Out;
   #Interlock_Horquilla.Horq_Out := #EstadoVI.Horq_Out;
   #EstadoVI.Horq_In := "ON" AND #Horq_In;
   #Interlock_Horquilla.Horq_In := #EstadoVI.Horq_In;
   #EstadoVI.Horq_EM_In := "ON" AND NOT #EM_Horq_In;
END_REGION

REGION Network 64: Salidas de la Horquilla
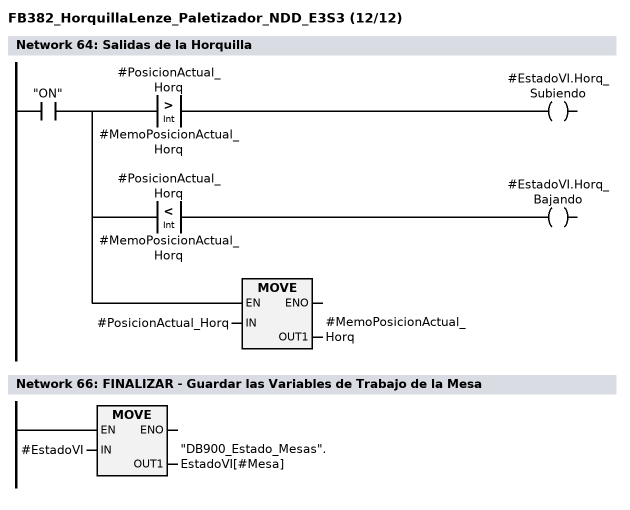
   RUNG wire#powerrail
      Contact( "ON" )
      wire#w1
      { S7_Templates := "SrcType := Int" } GT_Contact(in1 := #PosicionActual_Horq, in2 := #MemoPosicionActual_Horq)
      Coil( #EstadoVI.Horq_Subiendo )
   END_RUNG
   RUNG wire#w1
      { S7_Templates := "SrcType := Int" } LT_Contact(in1 := #PosicionActual_Horq, in2 := #MemoPosicionActual_Horq)
      Coil( #EstadoVI.Horq_Bajando )
   END_RUNG
   RUNG wire#w1
      Move(in := #PosicionActual_Horq, out1 => #MemoPosicionActual_Horq)
   END_RUNG
   // the same network as SCL:
   #EstadoVI.Horq_Subiendo := "ON" AND (#PosicionActual_Horq > #MemoPosicionActual_Horq);
   #EstadoVI.Horq_Bajando := "ON" AND (#PosicionActual_Horq < #MemoPosicionActual_Horq);
   IF "ON" THEN #MemoPosicionActual_Horq := #PosicionActual_Horq; END_IF;
END_REGION

REGION Network 65: ---
END_REGION

REGION Network 66: FINALIZAR - Guardar las Variables de Trabajo de la Mesa
   RUNG wire#powerrail
      Move(in := #EstadoVI, out1 => "DB900_Estado_Mesas".EstadoVI[#Mesa])
   END_RUNG
   // the same network as SCL:
   "DB900_Estado_Mesas".EstadoVI[#Mesa] := #EstadoVI;
END_REGION
END_FUNCTION_BLOCK
